LIN {X 0,Y 340.7,Z 163.546,A -85,B 0,C 180,E1 -14251.044,E2 -14251.044} C_VEL
LIN {X 0,Y 340.714,Z 163.527,A -85,B 0,C 180,E1 -14255.278,E2 -14255.278} C_VEL
LIN {X 0,Y 340.707,Z 163.544,A -85,B 0,C 180,E1 -14258.386,E2 -14258.386} C_VEL
LIN {X 0,Y 340.694,Z 163.543,A -85,B 0,C 180,E1 -14262.045,E2 -14262.045} C_VEL
LIN {X 0,Y 340.679,Z 163.532,A -85,B 0,C 180,E1 -14265.461,E2 -14265.461} C_VEL
LIN {X 0,Y 340.68,Z 163.504,A -85,B 0,C 180,E1 -14268.69,E2 -14268.69} C_VEL
LIN {X 0,Y 340.731,Z 163.543,A -85,B 0,C 180,E1 -14271.773,E2 -14271.773} C_VEL
LIN {X 0,Y 340.718,Z 163.515,A -85,B 0,C 180,E1 -14275.595,E2 -14275.595} C_VEL
LIN {X 0,Y 340.713,Z 163.54,A -85,B 0,C 180,E1 -14278.957,E2 -14278.957} C_VEL
LIN {X 0,Y 340.776,Z 163.536,A -85,B 0,C 180,E1 -14282.474,E2 -14282.474} C_VEL
LIN {X 0,Y 340.752,Z 163.541,A -85,B 0,C 180,E1 -14285.638,E2 -14285.638} C_VEL
LIN {X 0,Y 340.749,Z 163.652,A -85,B 0,C 180,E1 -14287.813,E2 -14287.813} C_VEL
LIN {X 0,Y 340.931,Z 164.489,A -85,B 0,C 180,E1 -14288.111,E2 -14288.111} C_VEL
LIN {X 0,Y 342.359,Z 167.226,A -85,B 0,C 180,E1 -14288.51,E2 -14288.51} C_VEL
LIN {X 0,Y 344.492,Z 169.253,A -85,B 0,C 180,E1 -14288.96,E2 -14288.96} C_VEL
LIN {X 0,Y 346.592,Z 172.469,A -85,B 0,C 180,E1 -14289.486,E2 -14289.486} C_VEL
LIN {X 0,Y 348.969,Z 174.84,A -85,B 0,C 180,E1 -14290.042,E2 -14290.042} C_VEL
LIN {X 0,Y 351.593,Z 178.193,A -85,B 0,C 180,E1 -14290.687,E2 -14290.687} C_VEL
LIN {X 0,Y 353.9,Z 180.47,A -85,B 0,C 180,E1 -14291.279,E2 -14291.279} C_VEL
LIN {X 0,Y 357.171,Z 184.318,A -85,B 0,C 180,E1 -14292.137,E2 -14292.137} C_VEL
LIN {X 0,Y 359.47,Z 186.421,A -85,B 0,C 180,E1 -14292.775,E2 -14292.775} C_VEL
LIN {X 0,Y 362.801,Z 190.102,A -85,B 0,C 180,E1 -14293.735,E2 -14293.735} C_VEL
LIN {X 0,Y 365.831,Z 192.588,A -85,B 0,C 180,E1 -14294.642,E2 -14294.642} C_VEL
LIN {X 0,Y 369.17,Z 196.334,A -85,B 0,C 180,E1 -14295.766,E2 -14295.766} C_VEL
LIN {X 0,Y 372.825,Z 199.259,A -85,B 0,C 180,E1 -14297.046,E2 -14297.046} C_VEL
LIN {X 0,Y 376.097,Z 202.708,A -85,B 0,C 180,E1 -14298.351,E2 -14298.351} C_VEL
LIN {X 0,Y 379.345,Z 205.079,A -85,B 0,C 180,E1 -14299.761,E2 -14299.761} C_VEL
LIN {X 0,Y 381.145,Z 206.14,A -85,B 0,C 180,E1 -14300.617,E2 -14300.617} C_VEL
LIN {X 0,Y 383.823,Z 209.323,A -85,B 0,C 180,E1 -14302.189,E2 -14302.189} C_VEL
LIN {X 0,Y 386.503,Z 211.375,A -85,B 0,C 180,E1 -14304.061,E2 -14304.061} C_VEL
LIN {X 0,Y 388.386,Z 212.415,A -85,B 0,C 180,E1 -14305.849,E2 -14305.849} C_VEL
LIN {X 0,Y 389.529,Z 212.797,A -85,B 0,C 180,E1 -14307.434,E2 -14307.434} C_VEL
LIN {X 0,Y 390.1,Z 213.221,A -85,B 0,C 180,E1 -14308.968,E2 -14308.968} C_VEL
LIN {X 0,Y 390.27,Z 213.15,A -85,B 0,C 180,E1 -14310,E2 -14310} C_VEL
LIN {X 0,Y 389.992,Z 213.112,A -85,B 0,C 180,E1 -14311.549,E2 -14311.549} C_VEL
LIN {X 0,Y 389.238,Z 212.653,A -85,B 0,C 180,E1 -14313.105,E2 -14313.105} C_VEL
LIN {X 0,Y 387.614,Z 212.058,A -85,B 0,C 180,E1 -14314.941,E2 -14314.941} C_VEL
LIN {X 0,Y 385.473,Z 210.702,A -85,B 0,C 180,E1 -14316.684,E2 -14316.684} C_VEL
LIN {X 0,Y 383.115,Z 208.634,A -85,B 0,C 180,E1 -14318.226,E2 -14318.226} C_VEL
LIN {X 0,Y 380.545,Z 205.669,A -85,B 0,C 180,E1 -14319.669,E2 -14319.669} C_VEL
LIN {X 0,Y 377.535,Z 203.906,A -85,B 0,C 180,E1 -14321.039,E2 -14321.039} C_VEL
LIN {X 0,Y 374.063,Z 200.682,A -85,B 0,C 180,E1 -14322.478,E2 -14322.478} C_VEL
LIN {X 0,Y 371.999,Z 198.446,A -85,B 0,C 180,E1 -14323.274,E2 -14323.274} C_VEL
LIN {X 0,Y 368.238,Z 195.449,A -85,B 0,C 180,E1 -14324.55,E2 -14324.55} C_VEL
LIN {X 0,Y 364.871,Z 191.735,A -85,B 0,C 180,E1 -14325.644,E2 -14325.644} C_VEL
LIN {X 0,Y 361.202,Z 188.491,A -85,B 0,C 180,E1 -14326.737,E2 -14326.737} C_VEL
LIN {X 0,Y 358.551,Z 185.445,A -85,B 0,C 180,E1 -14327.482,E2 -14327.482} C_VEL
LIN {X 0,Y 355.376,Z 182.455,A -85,B 0,C 180,E1 -14328.333,E2 -14328.333} C_VEL
LIN {X 0,Y 353.051,Z 179.523,A -85,B 0,C 180,E1 -14328.94,E2 -14328.94} C_VEL
LIN {X 0,Y 350.001,Z 176.372,A -85,B 0,C 180,E1 -14329.706,E2 -14329.706} C_VEL
LIN {X 0,Y 348.215,Z 173.968,A -85,B 0,C 180,E1 -14330.137,E2 -14330.137} C_VEL
LIN {X 0,Y 345.498,Z 171.058,A -85,B 0,C 180,E1 -14330.785,E2 -14330.785} C_VEL
LIN {X 0,Y 344.014,Z 168.683,A -85,B 0,C 180,E1 -14331.145,E2 -14331.145} C_VEL
LIN {X 0,Y 341.721,Z 166.358,A -85,B 0,C 180,E1 -14331.634,E2 -14331.634} C_VEL
LIN {X 0,Y 340.82,Z 164.079,A -85,B 0,C 180,E1 -14331.984,E2 -14331.984} C_VEL
LIN {X 0,Y 340.742,Z 163.555,A -85,B 0,C 180,E1 -14332.43,E2 -14332.43} C_VEL
LIN {X 0,Y 340.769,Z 163.54,A -85,B 0,C 180,E1 -14335.664,E2 -14335.664} C_VEL
LIN {X 0,Y 340.738,Z 163.528,A -85,B 0,C 180,E1 -14338.32,E2 -14338.32} C_VEL
LIN {X 0,Y 340.713,Z 163.54,A -85,B 0,C 180,E1 -14341.043,E2 -14341.043} C_VEL
LIN {X 0,Y 340.714,Z 163.517,A -85,B 0,C 180,E1 -14345.279,E2 -14345.279} C_VEL
LIN {X 0,Y 340.708,Z 163.547,A -85,B 0,C 180,E1 -14348.387,E2 -14348.387} C_VEL
LIN {X 0,Y 340.694,Z 163.499,A -85,B 0,C 180,E1 -14352.046,E2 -14352.046} C_VEL
LIN {X 0,Y 340.68,Z 163.546,A -85,B 0,C 180,E1 -14355.462,E2 -14355.462} C_VEL
LIN {X 0,Y 340.681,Z 163.536,A -85,B 0,C 180,E1 -14358.691,E2 -14358.691} C_VEL
LIN {X 0,Y 340.731,Z 163.541,A -85,B 0,C 180,E1 -14361.773,E2 -14361.773} C_VEL
LIN {X 0,Y 340.718,Z 163.522,A -85,B 0,C 180,E1 -14365.596,E2 -14365.596} C_VEL
LIN {X 0,Y 340.718,Z 163.542,A -85,B 0,C 180,E1 -14369.553,E2 -14369.553} C_VEL
LIN {X 0,Y 340.801,Z 163.511,A -85,B 0,C 180,E1 -14373.02,E2 -14373.02} C_VEL
LIN {X 0,Y 340.757,Z 163.528,A -85,B 0,C 180,E1 -14374.679,E2 -14374.679} C_VEL
LIN {X 0,Y 340.074,Z 163.621,A -85,B 0,C 180,E1 -14375.666,E2 -14375.666} C_VEL
LIN {X 0,Y 337.18,Z 163.982,A -85,B 0,C 180,E1 -14377.27,E2 -14377.27} C_VEL
LIN {X 0,Y 334.758,Z 164.276,A -85,B 0,C 180,E1 -14378.57,E2 -14378.57} C_VEL
LIN {X 0,Y 333.758,Z 164.391,A -85,B 0,C 180,E1 -14379.577,E2 -14379.577} C_VEL
LIN {X 0,Y 333.697,Z 164.392,A -85,B 0,C 180,E1 -14379.917,E2 -14379.917} C_VEL
LIN {X 0,Y 333.743,Z 164.401,A -85,B 0,C 180,E1 -14382.854,E2 -14382.854} C_VEL
LIN {X 0,Y 333.793,Z 164.402,A -85,B 0,C 180,E1 -14386.609,E2 -14386.609} C_VEL
LIN {X 0,Y 333.859,Z 164.366,A -85,B 0,C 180,E1 -14390.306,E2 -14390.306} C_VEL
LIN {X 0,Y 334.023,Z 164.369,A -85,B 0,C 180,E1 -14392.748,E2 -14392.748} C_VEL
LIN {X 0,Y 333.808,Z 164.403,A -85,B 0,C 180,E1 -14395.17,E2 -14395.17} C_VEL
LIN {X 0,Y 334.104,Z 164.352,A -85,B 0,C 180,E1 -14397.589,E2 -14397.589} C_VEL
LIN {X 0,Y 334.224,Z 164.319,A -85,B 0,C 180,E1 -14400.001,E2 -14400.001} C_VEL
LIN {X 0,Y 334.102,Z 164.359,A -85,B 0,C 180,E1 -14402.412,E2 -14402.412} C_VEL
LIN {X 0,Y 334.013,Z 164.374,A -85,B 0,C 180,E1 -14406.04,E2 -14406.04} C_VEL
LIN {X 0,Y 333.956,Z 164.361,A -85,B 0,C 180,E1 -14408.472,E2 -14408.472} C_VEL
LIN {X 0,Y 333.789,Z 164.397,A -85,B 0,C 180,E1 -14412.155,E2 -14412.155} C_VEL
LIN {X 0,Y 333.776,Z 164.399,A -85,B 0,C 180,E1 -14415.887,E2 -14415.887} C_VEL
LIN {X 0,Y 333.794,Z 164.375,A -85,B 0,C 180,E1 -14418.655,E2 -14418.655} C_VEL
LIN {X 0,Y 333.691,Z 164.414,A -85,B 0,C 180,E1 -14422.279,E2 -14422.279} C_VEL
LIN {X 0,Y 333.734,Z 164.392,A -85,B 0,C 180,E1 -14426.247,E2 -14426.247} C_VEL
LIN {X 0,Y 333.689,Z 164.41,A -85,B 0,C 180,E1 -14428.975,E2 -14428.975} C_VEL
LIN {X 0,Y 333.643,Z 164.416,A -85,B 0,C 180,E1 -14432.588,E2 -14432.588} C_VEL
LIN {X 0,Y 333.675,Z 164.415,A -85,B 0,C 180,E1 -14436.14,E2 -14436.14} C_VEL
LIN {X 0,Y 333.646,Z 164.414,A -85,B 0,C 180,E1 -14439.193,E2 -14439.193} C_VEL
LIN {X 0,Y 333.633,Z 164.429,A -85,B 0,C 180,E1 -14442.501,E2 -14442.501} C_VEL
LIN {X 0,Y 333.597,Z 164.429,A -85,B 0,C 180,E1 -14445.956,E2 -14445.956} C_VEL
LIN {X 0,Y 333.648,Z 164.399,A -85,B 0,C 180,E1 -14449.316,E2 -14449.316} C_VEL
LIN {X 0,Y 333.668,Z 164.417,A -85,B 0,C 180,E1 -14453.168,E2 -14453.168} C_VEL
LIN {X 0,Y 333.7,Z 164.494,A -85,B 0,C 180,E1 -14456.885,E2 -14456.885} C_VEL
LIN {X 0,Y 334.992,Z 170.834,A -85,B 0,C 180,E1 -14459.336,E2 -14459.336} C_VEL
LIN {X 0,Y 336.87,Z 180.369,A -85,B 0,C 180,E1 -14462.679,E2 -14462.679} C_VEL
LIN {X 0,Y 336.984,Z 184.304,A -85,B 0,C 180,E1 -14464.026,E2 -14464.026} C_VEL
LIN {X 0,Y 336.226,Z 190.3,A -85,B 0,C 180,E1 -14465.935,E2 -14465.935} C_VEL
LIN {X 0,Y 338.132,Z 199.11,A -85,B 0,C 180,E1 -14466.325,E2 -14466.325} C_VEL
LIN {X 0,Y 343.281,Z 226.363,A -85,B 0,C 180,E1 -14467.304,E2 -14467.304} C_VEL
LIN {X 0,Y 343.746,Z 230.733,A -85,B 0,C 180,E1 -14467.433,E2 -14467.433} C_VEL
LIN {X 0,Y 342.36,Z 296.356,A -85,B 0,C 180,E1 -14468.828,E2 -14468.828} C_VEL
LIN {X 0,Y 341.833,Z 306.667,A -85,B 0,C 180,E1 -14469.189,E2 -14469.189} C_VEL
LIN {X 0,Y 341.14,Z 316.179,A -85,B 0,C 180,E1 -14469.657,E2 -14469.657} C_VEL
LIN {X 0,Y 340.356,Z 325.253,A -85,B 0,C 180,E1 -14470.237,E2 -14470.237} C_VEL
LIN {X 0,Y 339.426,Z 334.384,A -85,B 0,C 180,E1 -14470.967,E2 -14470.967} C_VEL
LIN {X 0,Y 338.346,Z 343.378,A -85,B 0,C 180,E1 -14471.846,E2 -14471.846} C_VEL
LIN {X 0,Y 337.268,Z 352.105,A -85,B 0,C 180,E1 -14472.882,E2 -14472.882} C_VEL
LIN {X 0,Y 336.235,Z 360.291,A -85,B 0,C 180,E1 -14474.05,E2 -14474.05} C_VEL
LIN {X 0,Y 335.224,Z 368.347,A -85,B 0,C 180,E1 -14475.429,E2 -14475.429} C_VEL
LIN {X 0,Y 334.464,Z 374.299,A -85,B 0,C 180,E1 -14476.636,E2 -14476.636} C_VEL
LIN {X 0,Y 333.583,Z 380.614,A -85,B 0,C 180,E1 -14478.146,E2 -14478.146} C_VEL
LIN {X 0,Y 332.98,Z 385.877,A -85,B 0,C 180,E1 -14479.665,E2 -14479.665} C_VEL
LIN {X 0,Y 332.46,Z 391.008,A -85,B 0,C 180,E1 -14481.49,E2 -14481.49} C_VEL
LIN {X 0,Y 332.124,Z 394.996,A -85,B 0,C 180,E1 -14483.317,E2 -14483.317} C_VEL
LIN {X 0,Y 331.973,Z 397.946,A -85,B 0,C 180,E1 -14485.142,E2 -14485.142} C_VEL
LIN {X 0,Y 331.916,Z 400.393,A -85,B 0,C 180,E1 -14487.573,E2 -14487.573} C_VEL
LIN {X 0,Y 331.913,Z 400.982,A -85,B 0,C 180,E1 -14488.787,E2 -14488.787} C_VEL
LIN {X 0,Y 331.913,Z 400.982,A -85,B 0,C 180,E1 -14491.213,E2 -14491.213} C_VEL
LIN {X 0,Y 331.916,Z 400.393,A -85,B 0,C 180,E1 -14492.427,E2 -14492.427} C_VEL
LIN {X 0,Y 331.971,Z 397.946,A -85,B 0,C 180,E1 -14494.858,E2 -14494.858} C_VEL
LIN {X 0,Y 332.105,Z 394.996,A -85,B 0,C 180,E1 -14496.684,E2 -14496.684} C_VEL
LIN {X 0,Y 332.46,Z 391.008,A -85,B 0,C 180,E1 -14498.51,E2 -14498.51} C_VEL
LIN {X 0,Y 332.98,Z 385.877,A -85,B 0,C 180,E1 -14500.335,E2 -14500.335} C_VEL
LIN {X 0,Y 333.582,Z 380.614,A -85,B 0,C 180,E1 -14501.854,E2 -14501.854} C_VEL
LIN {X 0,Y 334.472,Z 374.299,A -85,B 0,C 180,E1 -14503.364,E2 -14503.364} C_VEL
LIN {X 0,Y 335.216,Z 368.347,A -85,B 0,C 180,E1 -14504.571,E2 -14504.571} C_VEL
LIN {X 0,Y 336.147,Z 361.42,A -85,B 0,C 180,E1 -14505.771,E2 -14505.771} C_VEL
LIN {X 0,Y 337.152,Z 353.24,A -85,B 0,C 180,E1 -14506.967,E2 -14506.967} C_VEL
LIN {X 0,Y 338.201,Z 344.73,A -85,B 0,C 180,E1 -14508.005,E2 -14508.005} C_VEL
LIN {X 0,Y 339.229,Z 336.016,A -85,B 0,C 180,E1 -14508.887,E2 -14508.887} C_VEL
LIN {X 0,Y 340.282,Z 326.26,A -85,B 0,C 180,E1 -14509.688,E2 -14509.688} C_VEL
LIN {X 0,Y 341.126,Z 316.179,A -85,B 0,C 180,E1 -14510.344,E2 -14510.344} C_VEL
LIN {X 0,Y 341.811,Z 306.666,A -85,B 0,C 180,E1 -14510.813,E2 -14510.813} C_VEL
LIN {X 0,Y 342.383,Z 296.357,A -85,B 0,C 180,E1 -14511.17,E2 -14511.17} C_VEL
LIN {X 0,Y 343.642,Z 228.699,A -85,B 0,C 180,E1 -14512.619,E2 -14512.619} C_VEL
LIN {X 0,Y 338.791,Z 202.108,A -85,B 0,C 180,E1 -14513.558,E2 -14513.558} C_VEL
LIN {X 0,Y 336.246,Z 190.61,A -85,B 0,C 180,E1 -14514.031,E2 -14514.031} C_VEL
LIN {X 0,Y 336.329,Z 189.001,A -85,B 0,C 180,E1 -14514.407,E2 -14514.407} C_VEL
LIN {X 0,Y 337.122,Z 183.29,A -85,B 0,C 180,E1 -14516.307,E2 -14516.307} C_VEL
LIN {X 0,Y 336.53,Z 178.586,A -85,B 0,C 180,E1 -14517.959,E2 -14517.959} C_VEL
LIN {X 0,Y 334.839,Z 169.883,A -85,B 0,C 180,E1 -14521.091,E2 -14521.091} C_VEL
LIN {X 0,Y 333.674,Z 164.43,A -85,B 0,C 180,E1 -14523.204,E2 -14523.204} C_VEL
LIN {X 0,Y 333.668,Z 164.417,A -85,B 0,C 180,E1 -14526.832,E2 -14526.832} C_VEL
LIN {X 0,Y 333.647,Z 164.399,A -85,B 0,C 180,E1 -14530.767,E2 -14530.767} C_VEL
LIN {X 0,Y 333.593,Z 164.428,A -85,B 0,C 180,E1 -14534.25,E2 -14534.25} C_VEL
LIN {X 0,Y 333.642,Z 164.428,A -85,B 0,C 180,E1 -14537.618,E2 -14537.618} C_VEL
LIN {X 0,Y 333.652,Z 164.416,A -85,B 0,C 180,E1 -14541.201,E2 -14541.201} C_VEL
LIN {X 0,Y 333.675,Z 164.415,A -85,B 0,C 180,E1 -14543.86,E2 -14543.86} C_VEL
LIN {X 0,Y 333.643,Z 164.416,A -85,B 0,C 180,E1 -14547.412,E2 -14547.412} C_VEL
LIN {X 0,Y 333.689,Z 164.41,A -85,B 0,C 180,E1 -14551.025,E2 -14551.025} C_VEL
LIN {X 0,Y 333.734,Z 164.392,A -85,B 0,C 180,E1 -14553.753,E2 -14553.753} C_VEL
LIN {X 0,Y 333.718,Z 164.411,A -85,B 0,C 180,E1 -14557.913,E2 -14557.913} C_VEL
LIN {X 0,Y 333.792,Z 164.376,A -85,B 0,C 180,E1 -14561.589,E2 -14561.589} C_VEL
LIN {X 0,Y 333.807,Z 164.401,A -85,B 0,C 180,E1 -14565.576,E2 -14565.576} C_VEL
LIN {X 0,Y 333.831,Z 164.375,A -85,B 0,C 180,E1 -14569.077,E2 -14569.077} C_VEL
LIN {X 0,Y 334.005,Z 164.366,A -85,B 0,C 180,E1 -14572.746,E2 -14572.746} C_VEL
LIN {X 0,Y 333.807,Z 164.403,A -85,B 0,C 180,E1 -14575.168,E2 -14575.168} C_VEL
LIN {X 0,Y 334.102,Z 164.359,A -85,B 0,C 180,E1 -14577.588,E2 -14577.588} C_VEL
LIN {X 0,Y 334.224,Z 164.319,A -85,B 0,C 180,E1 -14579.999,E2 -14579.999} C_VEL
LIN {X 0,Y 334.104,Z 164.352,A -85,B 0,C 180,E1 -14582.411,E2 -14582.411} C_VEL
LIN {X 0,Y 334.023,Z 164.369,A -85,B 0,C 180,E1 -14587.252,E2 -14587.252} C_VEL
LIN {X 0,Y 333.83,Z 164.376,A -85,B 0,C 180,E1 -14590.921,E2 -14590.921} C_VEL
LIN {X 0,Y 333.805,Z 164.404,A -85,B 0,C 180,E1 -14594.634,E2 -14594.634} C_VEL
LIN {X 0,Y 333.792,Z 164.376,A -85,B 0,C 180,E1 -14598.654,E2 -14598.654} C_VEL
LIN {X 0,Y 333.688,Z 164.419,A -85,B 0,C 180,E1 -14602.278,E2 -14602.278} C_VEL
LIN {X 0,Y 333.732,Z 164.395,A -85,B 0,C 180,E1 -14606.246,E2 -14606.246} C_VEL
LIN {X 0,Y 333.707,Z 164.406,A -85,B 0,C 180,E1 -14608.972,E2 -14608.972} C_VEL
LIN {X 0,Y 333.639,Z 164.421,A -85,B 0,C 180,E1 -14612.587,E2 -14612.587} C_VEL
LIN {X 0,Y 333.673,Z 164.417,A -85,B 0,C 180,E1 -14616.138,E2 -14616.138} C_VEL
LIN {X 0,Y 333.642,Z 164.419,A -85,B 0,C 180,E1 -14619.192,E2 -14619.192} C_VEL
LIN {X 0,Y 333.629,Z 164.424,A -85,B 0,C 180,E1 -14622.5,E2 -14622.5} C_VEL
LIN {X 0,Y 333.617,Z 164.404,A -85,B 0,C 180,E1 -14625.959,E2 -14625.959} C_VEL
LIN {X 0,Y 333.642,Z 164.388,A -85,B 0,C 180,E1 -14629.315,E2 -14629.315} C_VEL
LIN {X 0,Y 333.662,Z 164.416,A -85,B 0,C 180,E1 -14633.167,E2 -14633.167} C_VEL
LIN {X 0,Y 333.638,Z 164.409,A -85,B 0,C 180,E1 -14636.792,E2 -14636.792} C_VEL
LIN {X 0,Y 333.7,Z 164.403,A -85,B 0,C 180,E1 -14639.71,E2 -14639.71} C_VEL
LIN {X 0,Y 333.74,Z 164.411,A -85,B 0,C 180,E1 -14642.401,E2 -14642.401} C_VEL
LIN {X 0,Y 333.723,Z 164.417,A -85,B 0,C 180,E1 -14645.091,E2 -14645.091} C_VEL
LIN {X 0,Y 333.714,Z 164.564,A -85,B 0,C 180,E1 -14646.635,E2 -14646.635} C_VEL
LIN {X 0,Y 333.902,Z 165.477,A -85,B 0,C 180,E1 -14646.906,E2 -14646.906} C_VEL
LIN {X 0,Y 335.44,Z 168.254,A -85,B 0,C 180,E1 -14647.293,E2 -14647.293} C_VEL
LIN {X 0,Y 337.24,Z 170.143,A -85,B 0,C 180,E1 -14647.649,E2 -14647.649} C_VEL
LIN {X 0,Y 339.606,Z 173.544,A -85,B 0,C 180,E1 -14648.193,E2 -14648.193} C_VEL
LIN {X 0,Y 341.244,Z 175.293,A -85,B 0,C 180,E1 -14648.55,E2 -14648.55} C_VEL
LIN {X 0,Y 344.183,Z 179.022,A -85,B 0,C 180,E1 -14649.205,E2 -14649.205} C_VEL
LIN {X 0,Y 346.131,Z 181.092,A -85,B 0,C 180,E1 -14649.669,E2 -14649.669} C_VEL
LIN {X 0,Y 349.588,Z 185.013,A -85,B 0,C 180,E1 -14650.485,E2 -14650.485} C_VEL
LIN {X 0,Y 351.431,Z 186.973,A -85,B 0,C 180,E1 -14650.949,E2 -14650.949} C_VEL
LIN {X 0,Y 355.263,Z 191.068,A -85,B 0,C 180,E1 -14651.929,E2 -14651.929} C_VEL
LIN {X 0,Y 357.233,Z 192.994,A -85,B 0,C 180,E1 -14652.464,E2 -14652.464} C_VEL
LIN {X 0,Y 361.224,Z 197.042,A -85,B 0,C 180,E1 -14653.582,E2 -14653.582} C_VEL
LIN {X 0,Y 363.73,Z 199.166,A -85,B 0,C 180,E1 -14654.333,E2 -14654.333} C_VEL
LIN {X 0,Y 367.349,Z 202.937,A -85,B 0,C 180,E1 -14655.493,E2 -14655.493} C_VEL
LIN {X 0,Y 371.23,Z 206.057,A -85,B 0,C 180,E1 -14656.813,E2 -14656.813} C_VEL
LIN {X 0,Y 374.708,Z 209.566,A -85,B 0,C 180,E1 -14658.165,E2 -14658.165} C_VEL
LIN {X 0,Y 378.246,Z 212.061,A -85,B 0,C 180,E1 -14659.673,E2 -14659.673} C_VEL
LIN {X 0,Y 379.883,Z 213.156,A -85,B 0,C 180,E1 -14660.464,E2 -14660.464} C_VEL
LIN {X 0,Y 382.521,Z 216.119,A -85,B 0,C 180,E1 -14661.961,E2 -14661.961} C_VEL
LIN {X 0,Y 384.968,Z 218.058,A -85,B 0,C 180,E1 -14663.58,E2 -14663.58} C_VEL
LIN {X 0,Y 387.279,Z 219.357,A -85,B 0,C 180,E1 -14665.577,E2 -14665.577} C_VEL
LIN {X 0,Y 388.665,Z 219.823,A -85,B 0,C 180,E1 -14667.428,E2 -14667.428} C_VEL
LIN {X 0,Y 389.239,Z 220.26,A -85,B 0,C 180,E1 -14668.965,E2 -14668.965} C_VEL
LIN {X 0,Y 389.407,Z 220.18,A -85,B 0,C 180,E1 -14670,E2 -14670} C_VEL
LIN {X 0,Y 389.126,Z 220.135,A -85,B 0,C 180,E1 -14671.552,E2 -14671.552} C_VEL
LIN {X 0,Y 388.361,Z 219.7,A -85,B 0,C 180,E1 -14673.112,E2 -14673.112} C_VEL
LIN {X 0,Y 386.736,Z 219.095,A -85,B 0,C 180,E1 -14674.943,E2 -14674.943} C_VEL
LIN {X 0,Y 384.56,Z 217.784,A -85,B 0,C 180,E1 -14676.7,E2 -14676.7} C_VEL
LIN {X 0,Y 382.058,Z 215.691,A -85,B 0,C 180,E1 -14678.309,E2 -14678.309} C_VEL
LIN {X 0,Y 379.214,Z 212.563,A -85,B 0,C 180,E1 -14679.864,E2 -14679.864} C_VEL
LIN {X 0,Y 375.944,Z 210.617,A -85,B 0,C 180,E1 -14681.308,E2 -14681.308} C_VEL
LIN {X 0,Y 372.666,Z 207.666,A -85,B 0,C 180,E1 -14682.629,E2 -14682.629} C_VEL
LIN {X 0,Y 370.003,Z 204.947,A -85,B 0,C 180,E1 -14683.635,E2 -14683.635} C_VEL
LIN {X 0,Y 365.741,Z 201.421,A -85,B 0,C 180,E1 -14685.038,E2 -14685.038} C_VEL
LIN {X 0,Y 362.655,Z 198.154,A -85,B 0,C 180,E1 -14685.995,E2 -14685.995} C_VEL
LIN {X 0,Y 358.732,Z 194.722,A -85,B 0,C 180,E1 -14687.109,E2 -14687.109} C_VEL
LIN {X 0,Y 355.812,Z 191.514,A -85,B 0,C 180,E1 -14687.928,E2 -14687.928} C_VEL
LIN {X 0,Y 352.19,Z 187.976,A -85,B 0,C 180,E1 -14688.848,E2 -14688.848} C_VEL
LIN {X 0,Y 350.013,Z 185.387,A -85,B 0,C 180,E1 -14689.415,E2 -14689.415} C_VEL
LIN {X 0,Y 346.374,Z 181.474,A -85,B 0,C 180,E1 -14690.27,E2 -14690.27} C_VEL
LIN {X 0,Y 344.964,Z 179.746,A -85,B 0,C 180,E1 -14690.614,E2 -14690.614} C_VEL
LIN {X 0,Y 341.952,Z 176.423,A -85,B 0,C 180,E1 -14691.286,E2 -14691.286} C_VEL
LIN {X 0,Y 340.286,Z 174.152,A -85,B 0,C 180,E1 -14691.662,E2 -14691.662} C_VEL
LIN {X 0,Y 337.9,Z 171.309,A -85,B 0,C 180,E1 -14692.197,E2 -14692.197} C_VEL
LIN {X 0,Y 336.543,Z 169.281,A -85,B 0,C 180,E1 -14692.493,E2 -14692.493} C_VEL
LIN {X 0,Y 334.617,Z 167.13,A -85,B 0,C 180,E1 -14692.878,E2 -14692.878} C_VEL
LIN {X 0,Y 333.802,Z 165.071,A -85,B 0,C 180,E1 -14693.171,E2 -14693.171} C_VEL
LIN {X 0,Y 333.68,Z 164.493,A -85,B 0,C 180,E1 -14693.425,E2 -14693.425} C_VEL
LIN {X 0,Y 333.732,Z 164.416,A -85,B 0,C 180,E1 -14696.246,E2 -14696.246} C_VEL
LIN {X 0,Y 333.708,Z 164.397,A -85,B 0,C 180,E1 -14698.972,E2 -14698.972} C_VEL
LIN {X 0,Y 333.648,Z 164.418,A -85,B 0,C 180,E1 -14702.589,E2 -14702.589} C_VEL
LIN {X 0,Y 333.673,Z 164.405,A -85,B 0,C 180,E1 -14706.139,E2 -14706.139} C_VEL
LIN {X 0,Y 333.643,Z 164.418,A -85,B 0,C 180,E1 -14709.192,E2 -14709.192} C_VEL
LIN {X 0,Y 333.628,Z 164.379,A -85,B 0,C 180,E1 -14712.5,E2 -14712.5} C_VEL
LIN {X 0,Y 333.617,Z 164.426,A -85,B 0,C 180,E1 -14715.959,E2 -14715.959} C_VEL
LIN {X 0,Y 333.642,Z 164.41,A -85,B 0,C 180,E1 -14719.316,E2 -14719.316} C_VEL
LIN {X 0,Y 333.662,Z 164.42,A -85,B 0,C 180,E1 -14723.168,E2 -14723.168} C_VEL
LIN {X 0,Y 333.669,Z 164.4,A -85,B 0,C 180,E1 -14725.342,E2 -14725.342} C_VEL
LIN {X 0,Y 333.698,Z 164.417,A -85,B 0,C 180,E1 -14729.711,E2 -14729.711} C_VEL
LIN {X 0,Y 333.74,Z 164.39,A -85,B 0,C 180,E1 -14732.402,E2 -14732.402} C_VEL
LIN {X 0,Y 333.723,Z 164.411,A -85,B 0,C 180,E1 -14735.091,E2 -14735.091} C_VEL
LIN {X 0,Y 333.676,Z 164.409,A -85,B 0,C 180,E1 -14739.02,E2 -14739.02} C_VEL
LIN {X 0,Y 333.697,Z 164.392,A -85,B 0,C 180,E1 -14739.917,E2 -14739.917} C_VEL
LIN {X 0,Y 333.086,Z 164.465,A -85,B 0,C 180,E1 -14740.925,E2 -14740.925} C_VEL
LIN {X 0,Y 330.263,Z 164.828,A -85,B 0,C 180,E1 -14742.564,E2 -14742.564} C_VEL
LIN {X 0,Y 327.849,Z 165.141,A -85,B 0,C 180,E1 -14743.892,E2 -14743.892} C_VEL
LIN {X 0,Y 326.827,Z 165.273,A -85,B 0,C 180,E1 -14744.92,E2 -14744.92} C_VEL
LIN {X 0,Y 326.754,Z 165.282,A -85,B 0,C 180,E1 -14745.268,E2 -14745.268} C_VEL
LIN {X 0,Y 326.766,Z 165.259,A -85,B 0,C 180,E1 -14748.84,E2 -14748.84} C_VEL
LIN {X 0,Y 326.974,Z 165.247,A -85,B 0,C 180,E1 -14752.591,E2 -14752.591} C_VEL
LIN {X 0,Y 326.775,Z 165.279,A -85,B 0,C 180,E1 -14755.066,E2 -14755.066} C_VEL
LIN {X 0,Y 327.045,Z 165.231,A -85,B 0,C 180,E1 -14757.537,E2 -14757.537} C_VEL
LIN {X 0,Y 327.175,Z 165.196,A -85,B 0,C 180,E1 -14760.001,E2 -14760.001} C_VEL
LIN {X 0,Y 327.043,Z 165.238,A -85,B 0,C 180,E1 -14762.464,E2 -14762.464} C_VEL
LIN {X 0,Y 326.988,Z 165.248,A -85,B 0,C 180,E1 -14766.17,E2 -14766.17} C_VEL
LIN {X 0,Y 326.803,Z 165.243,A -85,B 0,C 180,E1 -14769.907,E2 -14769.907} C_VEL
LIN {X 0,Y 326.757,Z 165.28,A -85,B 0,C 180,E1 -14773.686,E2 -14773.686} C_VEL
LIN {X 0,Y 326.697,Z 165.264,A -85,B 0,C 180,E1 -14777.529,E2 -14777.529} C_VEL
LIN {X 0,Y 326.661,Z 165.275,A -85,B 0,C 180,E1 -14780.136,E2 -14780.136} C_VEL
LIN {X 0,Y 326.651,Z 165.291,A -85,B 0,C 180,E1 -14784.13,E2 -14784.13} C_VEL
LIN {X 0,Y 326.682,Z 165.267,A -85,B 0,C 180,E1 -14786.859,E2 -14786.859} C_VEL
LIN {X 0,Y 326.633,Z 165.299,A -85,B 0,C 180,E1 -14790.61,E2 -14790.61} C_VEL
LIN {X 0,Y 326.606,Z 165.281,A -85,B 0,C 180,E1 -14794.02,E2 -14794.02} C_VEL
LIN {X 0,Y 326.627,Z 165.299,A -85,B 0,C 180,E1 -14797.239,E2 -14797.239} C_VEL
LIN {X 0,Y 326.578,Z 165.298,A -85,B 0,C 180,E1 -14801.132,E2 -14801.132} C_VEL
LIN {X 0,Y 326.527,Z 165.303,A -85,B 0,C 180,E1 -14804.743,E2 -14804.743} C_VEL
LIN {X 0,Y 326.577,Z 165.292,A -85,B 0,C 180,E1 -14808.155,E2 -14808.155} C_VEL
LIN {X 0,Y 326.626,Z 165.289,A -85,B 0,C 180,E1 -14811.392,E2 -14811.392} C_VEL
LIN {X 0,Y 326.621,Z 165.284,A -85,B 0,C 180,E1 -14814.852,E2 -14814.852} C_VEL
LIN {X 0,Y 326.636,Z 165.412,A -85,B 0,C 180,E1 -14816.489,E2 -14816.489} C_VEL
LIN {X 0,Y 327.993,Z 171.946,A -85,B 0,C 180,E1 -14819.053,E2 -14819.053} C_VEL
LIN {X 0,Y 329.629,Z 180.163,A -85,B 0,C 180,E1 -14822.027,E2 -14822.027} C_VEL
LIN {X 0,Y 330.134,Z 184.112,A -85,B 0,C 180,E1 -14823.445,E2 -14823.445} C_VEL
LIN {X 0,Y 329.408,Z 189.966,A -85,B 0,C 180,E1 -14825.381,E2 -14825.381} C_VEL
LIN {X 0,Y 330.263,Z 194.285,A -85,B 0,C 180,E1 -14825.618,E2 -14825.618} C_VEL
LIN {X 0,Y 335.005,Z 217.321,A -85,B 0,C 180,E1 -14826.51,E2 -14826.51} C_VEL
LIN {X 0,Y 337.162,Z 230.559,A -85,B 0,C 180,E1 -14826.968,E2 -14826.968} C_VEL
LIN {X 0,Y 335.756,Z 296.164,A -85,B 0,C 180,E1 -14828.391,E2 -14828.391} C_VEL
LIN {X 0,Y 335.222,Z 306.475,A -85,B 0,C 180,E1 -14828.758,E2 -14828.758} C_VEL
LIN {X 0,Y 334.508,Z 315.988,A -85,B 0,C 180,E1 -14829.235,E2 -14829.235} C_VEL
LIN {X 0,Y 333.688,Z 325.061,A -85,B 0,C 180,E1 -14829.826,E2 -14829.826} C_VEL
LIN {X 0,Y 332.71,Z 334.193,A -85,B 0,C 180,E1 -14830.568,E2 -14830.568} C_VEL
LIN {X 0,Y 331.604,Z 343.186,A -85,B 0,C 180,E1 -14831.464,E2 -14831.464} C_VEL
LIN {X 0,Y 330.471,Z 351.913,A -85,B 0,C 180,E1 -14832.519,E2 -14832.519} C_VEL
LIN {X 0,Y 329.473,Z 359.673,A -85,B 0,C 180,E1 -14833.643,E2 -14833.643} C_VEL
LIN {X 0,Y 328.548,Z 366.662,A -85,B 0,C 180,E1 -14834.835,E2 -14834.835} C_VEL
LIN {X 0,Y 327.76,Z 372.731,A -85,B 0,C 180,E1 -14836.041,E2 -14836.041} C_VEL
LIN {X 0,Y 326.771,Z 379.266,A -85,B 0,C 180,E1 -14837.58,E2 -14837.58} C_VEL
LIN {X 0,Y 326.2,Z 383.768,A -85,B 0,C 180,E1 -14838.819,E2 -14838.819} C_VEL
LIN {X 0,Y 325.572,Z 389.261,A -85,B 0,C 180,E1 -14840.683,E2 -14840.683} C_VEL
LIN {X 0,Y 325.153,Z 393.587,A -85,B 0,C 180,E1 -14842.549,E2 -14842.549} C_VEL
LIN {X 0,Y 324.925,Z 396.619,A -85,B 0,C 180,E1 -14844.251,E2 -14844.251} C_VEL
LIN {X 0,Y 324.876,Z 399.144,A -85,B 0,C 180,E1 -14846.279,E2 -14846.279} C_VEL
LIN {X 0,Y 324.835,Z 400.202,A -85,B 0,C 180,E1 -14847.52,E2 -14847.52} C_VEL
LIN {X 0,Y 324.822,Z 400.791,A -85,B 0,C 180,E1 -14848.76,E2 -14848.76} C_VEL
LIN {X 0,Y 324.822,Z 400.791,A -85,B 0,C 180,E1 -14851.24,E2 -14851.24} C_VEL
LIN {X 0,Y 324.835,Z 400.202,A -85,B 0,C 180,E1 -14852.48,E2 -14852.48} C_VEL
LIN {X 0,Y 324.881,Z 397.754,A -85,B 0,C 180,E1 -14854.964,E2 -14854.964} C_VEL
LIN {X 0,Y 325.047,Z 394.804,A -85,B 0,C 180,E1 -14856.83,E2 -14856.83} C_VEL
LIN {X 0,Y 325.4,Z 390.815,A -85,B 0,C 180,E1 -14858.696,E2 -14858.696} C_VEL
LIN {X 0,Y 325.959,Z 385.684,A -85,B 0,C 180,E1 -14860.56,E2 -14860.56} C_VEL
LIN {X 0,Y 326.617,Z 380.422,A -85,B 0,C 180,E1 -14862.11,E2 -14862.11} C_VEL
LIN {X 0,Y 327.554,Z 374.107,A -85,B 0,C 180,E1 -14863.651,E2 -14863.651} C_VEL
LIN {X 0,Y 328.32,Z 368.154,A -85,B 0,C 180,E1 -14864.884,E2 -14864.884} C_VEL
LIN {X 0,Y 329.28,Z 361.228,A -85,B 0,C 180,E1 -14866.109,E2 -14866.109} C_VEL
LIN {X 0,Y 330.325,Z 353.047,A -85,B 0,C 180,E1 -14867.329,E2 -14867.329} C_VEL
LIN {X 0,Y 331.458,Z 344.538,A -85,B 0,C 180,E1 -14868.385,E2 -14868.385} C_VEL
LIN {X 0,Y 332.516,Z 335.824,A -85,B 0,C 180,E1 -14869.284,E2 -14869.284} C_VEL
LIN {X 0,Y 333.603,Z 326.068,A -85,B 0,C 180,E1 -14870.099,E2 -14870.099} C_VEL
LIN {X 0,Y 334.473,Z 315.987,A -85,B 0,C 180,E1 -14870.767,E2 -14870.767} C_VEL
LIN {X 0,Y 335.198,Z 306.475,A -85,B 0,C 180,E1 -14871.243,E2 -14871.243} C_VEL
LIN {X 0,Y 335.778,Z 296.165,A -85,B 0,C 180,E1 -14871.607,E2 -14871.607} C_VEL
LIN {X 0,Y 337.131,Z 230.29,A -85,B 0,C 180,E1 -14873.041,E2 -14873.041} C_VEL
LIN {X 0,Y 333.079,Z 207.235,A -85,B 0,C 180,E1 -14873.865,E2 -14873.865} C_VEL
LIN {X 0,Y 329.433,Z 190.195,A -85,B 0,C 180,E1 -14874.582,E2 -14874.582} C_VEL
LIN {X 0,Y 329.641,Z 187.957,A -85,B 0,C 180,E1 -14875.239,E2 -14875.239} C_VEL
LIN {X 0,Y 330.155,Z 183.942,A -85,B 0,C 180,E1 -14876.612,E2 -14876.612} C_VEL
LIN {X 0,Y 328.872,Z 176.177,A -85,B 0,C 180,E1 -14879.44,E2 -14879.44} C_VEL
LIN {X 0,Y 326.906,Z 166.644,A -85,B 0,C 180,E1 -14883.023,E2 -14883.023} C_VEL
LIN {X 0,Y 326.626,Z 165.314,A -85,B 0,C 180,E1 -14883.584,E2 -14883.584} C_VEL
LIN {X 0,Y 326.631,Z 165.298,A -85,B 0,C 180,E1 -14887.238,E2 -14887.238} C_VEL
LIN {X 0,Y 326.578,Z 165.282,A -85,B 0,C 180,E1 -14891.13,E2 -14891.13} C_VEL
LIN {X 0,Y 326.527,Z 165.306,A -85,B 0,C 180,E1 -14894.742,E2 -14894.742} C_VEL
LIN {X 0,Y 326.576,Z 165.304,A -85,B 0,C 180,E1 -14898.153,E2 -14898.153} C_VEL
LIN {X 0,Y 326.623,Z 165.294,A -85,B 0,C 180,E1 -14901.391,E2 -14901.391} C_VEL
LIN {X 0,Y 326.619,Z 165.286,A -85,B 0,C 180,E1 -14904.851,E2 -14904.851} C_VEL
LIN {X 0,Y 326.607,Z 165.292,A -85,B 0,C 180,E1 -14907.455,E2 -14907.455} C_VEL
LIN {X 0,Y 326.647,Z 165.294,A -85,B 0,C 180,E1 -14910.339,E2 -14910.339} C_VEL
LIN {X 0,Y 326.689,Z 165.275,A -85,B 0,C 180,E1 -14914.515,E2 -14914.515} C_VEL
LIN {X 0,Y 326.644,Z 165.29,A -85,B 0,C 180,E1 -14918.544,E2 -14918.544} C_VEL
LIN {X 0,Y 326.743,Z 165.252,A -85,B 0,C 180,E1 -14921.177,E2 -14921.177} C_VEL
LIN {X 0,Y 326.761,Z 165.279,A -85,B 0,C 180,E1 -14925.432,E2 -14925.432} C_VEL
LIN {X 0,Y 326.767,Z 165.257,A -85,B 0,C 180,E1 -14928.838,E2 -14928.838} C_VEL
LIN {X 0,Y 326.957,Z 165.242,A -85,B 0,C 180,E1 -14932.589,E2 -14932.589} C_VEL
LIN {X 0,Y 326.774,Z 165.28,A -85,B 0,C 180,E1 -14935.064,E2 -14935.064} C_VEL
LIN {X 0,Y 327.043,Z 165.238,A -85,B 0,C 180,E1 -14937.536,E2 -14937.536} C_VEL
LIN {X 0,Y 327.175,Z 165.196,A -85,B 0,C 180,E1 -14939.999,E2 -14939.999} C_VEL
LIN {X 0,Y 327.045,Z 165.231,A -85,B 0,C 180,E1 -14942.463,E2 -14942.463} C_VEL
LIN {X 0,Y 326.968,Z 165.249,A -85,B 0,C 180,E1 -14946.644,E2 -14946.644} C_VEL
LIN {X 0,Y 326.81,Z 165.243,A -85,B 0,C 180,E1 -14949.906,E2 -14949.906} C_VEL
LIN {X 0,Y 326.755,Z 165.28,A -85,B 0,C 180,E1 -14953.685,E2 -14953.685} C_VEL
LIN {X 0,Y 326.695,Z 165.271,A -85,B 0,C 180,E1 -14957.527,E2 -14957.527} C_VEL
LIN {X 0,Y 326.658,Z 165.27,A -85,B 0,C 180,E1 -14960.134,E2 -14960.134} C_VEL
LIN {X 0,Y 326.648,Z 165.294,A -85,B 0,C 180,E1 -14964.128,E2 -14964.128} C_VEL
LIN {X 0,Y 326.681,Z 165.269,A -85,B 0,C 180,E1 -14966.857,E2 -14966.857} C_VEL
LIN {X 0,Y 326.635,Z 165.297,A -85,B 0,C 180,E1 -14970.611,E2 -14970.611} C_VEL
LIN {X 0,Y 326.602,Z 165.281,A -85,B 0,C 180,E1 -14974.019,E2 -14974.019} C_VEL
LIN {X 0,Y 326.625,Z 165.3,A -85,B 0,C 180,E1 -14977.239,E2 -14977.239} C_VEL
LIN {X 0,Y 326.573,Z 165.291,A -85,B 0,C 180,E1 -14981.131,E2 -14981.131} C_VEL
LIN {X 0,Y 326.552,Z 165.301,A -85,B 0,C 180,E1 -14984.748,E2 -14984.748} C_VEL
LIN {X 0,Y 326.571,Z 165.256,A -85,B 0,C 180,E1 -14988.154,E2 -14988.154} C_VEL
LIN {X 0,Y 326.62,Z 165.3,A -85,B 0,C 180,E1 -14991.391,E2 -14991.391} C_VEL
LIN {X 0,Y 326.615,Z 165.271,A -85,B 0,C 180,E1 -14994.851,E2 -14994.851} C_VEL
LIN {X 0,Y 326.612,Z 165.295,A -85,B 0,C 180,E1 -14997.456,E2 -14997.456} C_VEL
LIN {X 0,Y 326.658,Z 165.275,A -85,B 0,C 180,E1 -15000.341,E2 -15000.341} C_VEL
LIN {X 0,Y 326.686,Z 165.294,A -85,B 0,C 180,E1 -15004.516,E2 -15004.516} C_VEL
LIN {X 0,Y 326.691,Z 165.587,A -85,B 0,C 180,E1 -15005.621,E2 -15005.621} C_VEL
LIN {X 0,Y 326.997,Z 166.824,A -85,B 0,C 180,E1 -15005.854,E2 -15005.854} C_VEL
LIN {X 0,Y 328.544,Z 169.353,A -85,B 0,C 180,E1 -15006.172,E2 -15006.172} C_VEL
LIN {X 0,Y 329.922,Z 170.862,A -85,B 0,C 180,E1 -15006.429,E2 -15006.429} C_VEL
LIN {X 0,Y 332.332,Z 174.357,A -85,B 0,C 180,E1 -15006.946,E2 -15006.946} C_VEL
LIN {X 0,Y 333.847,Z 176.146,A -85,B 0,C 180,E1 -15007.255,E2 -15007.255} C_VEL
LIN {X 0,Y 336.858,Z 179.834,A -85,B 0,C 180,E1 -15007.873,E2 -15007.873} C_VEL
LIN {X 0,Y 341.329,Z 185.197,A -85,B 0,C 180,E1 -15008.866,E2 -15008.866} C_VEL
LIN {X 0,Y 343.578,Z 187.673,A -85,B 0,C 180,E1 -15009.36,E2 -15009.36} C_VEL
LIN {X 0,Y 347.347,Z 191.645,A -85,B 0,C 180,E1 -15010.249,E2 -15010.249} C_VEL
LIN {X 0,Y 352.203,Z 196.917,A -85,B 0,C 180,E1 -15011.455,E2 -15011.455} C_VEL
LIN {X 0,Y 354.866,Z 199.388,A -85,B 0,C 180,E1 -15012.126,E2 -15012.126} C_VEL
LIN {X 0,Y 359.165,Z 203.614,A -85,B 0,C 180,E1 -15013.306,E2 -15013.306} C_VEL
LIN {X 0,Y 361.621,Z 205.668,A -85,B 0,C 180,E1 -15014.013,E2 -15014.013} C_VEL
LIN {X 0,Y 365.635,Z 209.686,A -85,B 0,C 180,E1 -15015.257,E2 -15015.257} C_VEL
LIN {X 0,Y 369.613,Z 212.872,A -85,B 0,C 180,E1 -15016.584,E2 -15016.584} C_VEL
LIN {X 0,Y 373.669,Z 216.74,A -85,B 0,C 180,E1 -15018.131,E2 -15018.131} C_VEL
LIN {X 0,Y 377.405,Z 219.212,A -85,B 0,C 180,E1 -15019.711,E2 -15019.711} C_VEL
LIN {X 0,Y 378.641,Z 220.158,A -85,B 0,C 180,E1 -15020.316,E2 -15020.316} C_VEL
LIN {X 0,Y 381.246,Z 222.96,A -85,B 0,C 180,E1 -15021.75,E2 -15021.75} C_VEL
LIN {X 0,Y 383.646,Z 224.871,A -85,B 0,C 180,E1 -15023.284,E2 -15023.284} C_VEL
LIN {X 0,Y 385.845,Z 226.138,A -85,B 0,C 180,E1 -15025.046,E2 -15025.046} C_VEL
LIN {X 0,Y 387.489,Z 226.713,A -85,B 0,C 180,E1 -15026.881,E2 -15026.881} C_VEL
LIN {X 0,Y 388.378,Z 227.295,A -85,B 0,C 180,E1 -15028.963,E2 -15028.963} C_VEL
LIN {X 0,Y 388.542,Z 227.227,A -85,B 0,C 180,E1 -15030,E2 -15030} C_VEL
LIN {X 0,Y 388.258,Z 227.183,A -85,B 0,C 180,E1 -15031.556,E2 -15031.556} C_VEL
LIN {X 0,Y 387.234,Z 226.669,A -85,B 0,C 180,E1 -15033.443,E2 -15033.443} C_VEL
LIN {X 0,Y 385.526,Z 225.999,A -85,B 0,C 180,E1 -15035.23,E2 -15035.23} C_VEL
LIN {X 0,Y 383.278,Z 224.592,A -85,B 0,C 180,E1 -15036.977,E2 -15036.977} C_VEL
LIN {X 0,Y 380.599,Z 222.31,A -85,B 0,C 180,E1 -15038.639,E2 -15038.639} C_VEL
LIN {X 0,Y 377.888,Z 219.451,A -85,B 0,C 180,E1 -15040.06,E2 -15040.06} C_VEL
LIN {X 0,Y 374.225,Z 217.199,A -85,B 0,C 180,E1 -15041.637,E2 -15041.637} C_VEL
LIN {X 0,Y 370.283,Z 213.606,A -85,B 0,C 180,E1 -15043.165,E2 -15043.165} C_VEL
LIN {X 0,Y 368.107,Z 211.584,A -85,B 0,C 180,E1 -15043.926,E2 -15043.926} C_VEL
LIN {X 0,Y 363.709,Z 207.954,A -85,B 0,C 180,E1 -15045.342,E2 -15045.342} C_VEL
LIN {X 0,Y 360.454,Z 204.596,A -85,B 0,C 180,E1 -15046.334,E2 -15046.334} C_VEL
LIN {X 0,Y 355.913,Z 200.562,A -85,B 0,C 180,E1 -15047.589,E2 -15047.589} C_VEL
LIN {X 0,Y 353.163,Z 197.706,A -85,B 0,C 180,E1 -15048.309,E2 -15048.309} C_VEL
LIN {X 0,Y 349.304,Z 193.886,A -85,B 0,C 180,E1 -15049.284,E2 -15049.284} C_VEL
LIN {X 0,Y 346.286,Z 190.674,A -85,B 0,C 180,E1 -15049.994,E2 -15049.994} C_VEL
LIN {X 0,Y 342.731,Z 186.542,A -85,B 0,C 180,E1 -15050.838,E2 -15050.838} C_VEL
LIN {X 0,Y 338.478,Z 181.938,A -85,B 0,C 180,E1 -15051.76,E2 -15051.76} C_VEL
LIN {X 0,Y 336.613,Z 179.601,A -85,B 0,C 180,E1 -15052.177,E2 -15052.177} C_VEL
LIN {X 0,Y 333.567,Z 175.716,A -85,B 0,C 180,E1 -15052.804,E2 -15052.804} C_VEL
LIN {X 0,Y 330.474,Z 171.844,A -85,B 0,C 180,E1 -15053.45,E2 -15053.45} C_VEL
LIN {X 0,Y 329.168,Z 169.925,A -85,B 0,C 180,E1 -15053.716,E2 -15053.716} C_VEL
LIN {X 0,Y 327.268,Z 167.481,A -85,B 0,C 180,E1 -15054.08,E2 -15054.08} C_VEL
LIN {X 0,Y 326.717,Z 165.742,A -85,B 0,C 180,E1 -15054.335,E2 -15054.335} C_VEL
LIN {X 0,Y 326.684,Z 165.294,A -85,B 0,C 180,E1 -15054.803,E2 -15054.803} C_VEL
LIN {X 0,Y 326.653,Z 165.281,A -85,B 0,C 180,E1 -15058.251,E2 -15058.251} C_VEL
LIN {X 0,Y 326.598,Z 165.299,A -85,B 0,C 180,E1 -15061.094,E2 -15061.094} C_VEL
LIN {X 0,Y 326.605,Z 165.273,A -85,B 0,C 180,E1 -15064.019,E2 -15064.019} C_VEL
LIN {X 0,Y 326.625,Z 165.297,A -85,B 0,C 180,E1 -15067.239,E2 -15067.239} C_VEL
LIN {X 0,Y 326.572,Z 165.261,A -85,B 0,C 180,E1 -15071.131,E2 -15071.131} C_VEL
LIN {X 0,Y 326.552,Z 165.293,A -85,B 0,C 180,E1 -15074.748,E2 -15074.748} C_VEL
LIN {X 0,Y 326.572,Z 165.299,A -85,B 0,C 180,E1 -15078.155,E2 -15078.155} C_VEL
LIN {X 0,Y 326.62,Z 165.299,A -85,B 0,C 180,E1 -15081.392,E2 -15081.392} C_VEL
LIN {X 0,Y 326.615,Z 165.281,A -85,B 0,C 180,E1 -15084.852,E2 -15084.852} C_VEL
LIN {X 0,Y 326.603,Z 165.298,A -85,B 0,C 180,E1 -15087.456,E2 -15087.456} C_VEL
LIN {X 0,Y 326.656,Z 165.29,A -85,B 0,C 180,E1 -15090.341,E2 -15090.341} C_VEL
LIN {X 0,Y 326.686,Z 165.28,A -85,B 0,C 180,E1 -15094.517,E2 -15094.517} C_VEL
LIN {X 0,Y 326.642,Z 165.287,A -85,B 0,C 180,E1 -15098.546,E2 -15098.546} C_VEL
LIN {X 0,Y 326.741,Z 165.253,A -85,B 0,C 180,E1 -15101.178,E2 -15101.178} C_VEL
LIN {X 0,Y 326.754,Z 165.282,A -85,B 0,C 180,E1 -15105.268,E2 -15105.268} C_VEL
LIN {X 0,Y 326.103,Z 165.363,A -85,B 0,C 180,E1 -15106.297,E2 -15106.297} C_VEL
LIN {X 0,Y 323.239,Z 165.705,A -85,B 0,C 180,E1 -15107.971,E2 -15107.971} C_VEL
LIN {X 0,Y 320.832,Z 165.991,A -85,B 0,C 180,E1 -15109.328,E2 -15109.328} C_VEL
LIN {X 0,Y 319.847,Z 166.11,A -85,B 0,C 180,E1 -15110.379,E2 -15110.379} C_VEL
LIN {X 0,Y 319.794,Z 166.118,A -85,B 0,C 180,E1 -15110.734,E2 -15110.734} C_VEL
LIN {X 0,Y 319.949,Z 166.127,A -85,B 0,C 180,E1 -15113.695,E2 -15113.695} C_VEL
LIN {X 0,Y 319.988,Z 166.111,A -85,B 0,C 180,E1 -15117.483,E2 -15117.483} C_VEL
LIN {X 0,Y 320.128,Z 166.073,A -85,B 0,C 180,E1 -15120.001,E2 -15120.001} C_VEL
LIN {X 0,Y 319.987,Z 166.117,A -85,B 0,C 180,E1 -15122.518,E2 -15122.518} C_VEL
LIN {X 0,Y 319.942,Z 166.126,A -85,B 0,C 180,E1 -15126.306,E2 -15126.306} C_VEL
LIN {X 0,Y 319.835,Z 166.113,A -85,B 0,C 180,E1 -15128.849,E2 -15128.849} C_VEL
LIN {X 0,Y 319.679,Z 166.155,A -85,B 0,C 180,E1 -15132.701,E2 -15132.701} C_VEL
LIN {X 0,Y 319.698,Z 166.157,A -85,B 0,C 180,E1 -15135.296,E2 -15135.296} C_VEL
LIN {X 0,Y 319.673,Z 166.134,A -85,B 0,C 180,E1 -15139.256,E2 -15139.256} C_VEL
LIN {X 0,Y 319.569,Z 166.176,A -85,B 0,C 180,E1 -15143.32,E2 -15143.32} C_VEL
LIN {X 0,Y 319.633,Z 166.148,A -85,B 0,C 180,E1 -15146.089,E2 -15146.089} C_VEL
LIN {X 0,Y 319.579,Z 166.166,A -85,B 0,C 180,E1 -15148.935,E2 -15148.935} C_VEL
LIN {X 0,Y 319.53,Z 166.18,A -85,B 0,C 180,E1 -15151.863,E2 -15151.863} C_VEL
LIN {X 0,Y 319.579,Z 166.167,A -85,B 0,C 180,E1 -15155.544,E2 -15155.544} C_VEL
LIN {X 0,Y 319.572,Z 166.177,A -85,B 0,C 180,E1 -15158.009,E2 -15158.009} C_VEL
LIN {X 0,Y 319.526,Z 166.18,A -85,B 0,C 180,E1 -15161.598,E2 -15161.598} C_VEL
LIN {X 0,Y 319.488,Z 166.182,A -85,B 0,C 180,E1 -15165.258,E2 -15165.258} C_VEL
LIN {X 0,Y 319.529,Z 166.162,A -85,B 0,C 180,E1 -15168.712,E2 -15168.712} C_VEL
LIN {X 0,Y 319.58,Z 166.18,A -85,B 0,C 180,E1 -15172.345,E2 -15172.345} C_VEL
LIN {X 0,Y 319.59,Z 166.289,A -85,B 0,C 180,E1 -15176.049,E2 -15176.049} C_VEL
LIN {X 0,Y 320.964,Z 172.754,A -85,B 0,C 180,E1 -15178.647,E2 -15178.647} C_VEL
LIN {X 0,Y 322.75,Z 181.936,A -85,B 0,C 180,E1 -15182.085,E2 -15182.085} C_VEL
LIN {X 0,Y 323.075,Z 186.232,A -85,B 0,C 180,E1 -15183.654,E2 -15183.654} C_VEL
LIN {X 0,Y 322.586,Z 189.926,A -85,B 0,C 180,E1 -15184.85,E2 -15184.85} C_VEL
LIN {X 0,Y 324.838,Z 200.086,A -85,B 0,C 180,E1 -15185.326,E2 -15185.326} C_VEL
LIN {X 0,Y 329.604,Z 224.903,A -85,B 0,C 180,E1 -15186.281,E2 -15186.281} C_VEL
LIN {X 0,Y 330.622,Z 232.075,A -85,B 0,C 180,E1 -15186.524,E2 -15186.524} C_VEL
LIN {X 0,Y 329.18,Z 295.973,A -85,B 0,C 180,E1 -15187.937,E2 -15187.937} C_VEL
LIN {X 0,Y 328.628,Z 306.284,A -85,B 0,C 180,E1 -15188.311,E2 -15188.311} C_VEL
LIN {X 0,Y 327.873,Z 315.796,A -85,B 0,C 180,E1 -15188.795,E2 -15188.795} C_VEL
LIN {X 0,Y 327.027,Z 324.869,A -85,B 0,C 180,E1 -15189.396,E2 -15189.396} C_VEL
LIN {X 0,Y 326.021,Z 334.001,A -85,B 0,C 180,E1 -15190.153,E2 -15190.153} C_VEL
LIN {X 0,Y 324.884,Z 342.995,A -85,B 0,C 180,E1 -15191.066,E2 -15191.066} C_VEL
LIN {X 0,Y 323.698,Z 351.721,A -85,B 0,C 180,E1 -15192.141,E2 -15192.141} C_VEL
LIN {X 0,Y 322.681,Z 359.115,A -85,B 0,C 180,E1 -15193.227,E2 -15193.227} C_VEL
LIN {X 0,Y 321.657,Z 366.643,A -85,B 0,C 180,E1 -15194.537,E2 -15194.537} C_VEL
LIN {X 0,Y 320.843,Z 372.539,A -85,B 0,C 180,E1 -15195.734,E2 -15195.734} C_VEL
LIN {X 0,Y 319.824,Z 379.074,A -85,B 0,C 180,E1 -15197.306,E2 -15197.306} C_VEL
LIN {X 0,Y 319.19,Z 383.575,A -85,B 0,C 180,E1 -15198.571,E2 -15198.571} C_VEL
LIN {X 0,Y 318.538,Z 389.069,A -85,B 0,C 180,E1 -15200.475,E2 -15200.475} C_VEL
LIN {X 0,Y 318.077,Z 393.394,A -85,B 0,C 180,E1 -15202.382,E2 -15202.382} C_VEL
LIN {X 0,Y 317.839,Z 396.666,A -85,B 0,C 180,E1 -15204.291,E2 -15204.291} C_VEL
LIN {X 0,Y 317.786,Z 398.952,A -85,B 0,C 180,E1 -15206.196,E2 -15206.196} C_VEL
LIN {X 0,Y 317.756,Z 400.011,A -85,B 0,C 180,E1 -15207.465,E2 -15207.465} C_VEL
LIN {X 0,Y 317.734,Z 400.599,A -85,B 0,C 180,E1 -15208.733,E2 -15208.733} C_VEL
LIN {X 0,Y 317.734,Z 400.599,A -85,B 0,C 180,E1 -15211.267,E2 -15211.267} C_VEL
LIN {X 0,Y 317.756,Z 400.011,A -85,B 0,C 180,E1 -15212.535,E2 -15212.535} C_VEL
LIN {X 0,Y 317.796,Z 397.562,A -85,B 0,C 180,E1 -15215.075,E2 -15215.075} C_VEL
LIN {X 0,Y 317.985,Z 394.612,A -85,B 0,C 180,E1 -15216.982,E2 -15216.982} C_VEL
LIN {X 0,Y 318.361,Z 390.623,A -85,B 0,C 180,E1 -15218.889,E2 -15218.889} C_VEL
LIN {X 0,Y 318.948,Z 385.492,A -85,B 0,C 180,E1 -15220.795,E2 -15220.795} C_VEL
LIN {X 0,Y 319.63,Z 380.229,A -85,B 0,C 180,E1 -15222.379,E2 -15222.379} C_VEL
LIN {X 0,Y 320.629,Z 373.914,A -85,B 0,C 180,E1 -15223.952,E2 -15223.952} C_VEL
LIN {X 0,Y 321.444,Z 367.962,A -85,B 0,C 180,E1 -15225.21,E2 -15225.21} C_VEL
LIN {X 0,Y 322.41,Z 361.034,A -85,B 0,C 180,E1 -15226.462,E2 -15226.462} C_VEL
LIN {X 0,Y 323.54,Z 352.855,A -85,B 0,C 180,E1 -15227.704,E2 -15227.704} C_VEL
LIN {X 0,Y 324.725,Z 344.346,A -85,B 0,C 180,E1 -15228.78,E2 -15228.78} C_VEL
LIN {X 0,Y 325.804,Z 335.632,A -85,B 0,C 180,E1 -15229.697,E2 -15229.697} C_VEL
LIN {X 0,Y 326.949,Z 325.877,A -85,B 0,C 180,E1 -15230.527,E2 -15230.527} C_VEL
LIN {X 0,Y 327.853,Z 315.796,A -85,B 0,C 180,E1 -15231.207,E2 -15231.207} C_VEL
LIN {X 0,Y 328.58,Z 306.283,A -85,B 0,C 180,E1 -15231.692,E2 -15231.692} C_VEL
LIN {X 0,Y 329.193,Z 295.974,A -85,B 0,C 180,E1 -15232.062,E2 -15232.062} C_VEL
LIN {X 0,Y 330.599,Z 231.386,A -85,B 0,C 180,E1 -15233.493,E2 -15233.493} C_VEL
LIN {X 0,Y 326.809,Z 209.434,A -85,B 0,C 180,E1 -15234.296,E2 -15234.296} C_VEL
LIN {X 0,Y 322.619,Z 190.102,A -85,B 0,C 180,E1 -15235.127,E2 -15235.127} C_VEL
LIN {X 0,Y 322.726,Z 188.615,A -85,B 0,C 180,E1 -15235.508,E2 -15235.508} C_VEL
LIN {X 0,Y 323.131,Z 184.669,A -85,B 0,C 180,E1 -15236.906,E2 -15236.906} C_VEL
LIN {X 0,Y 321.927,Z 177.478,A -85,B 0,C 180,E1 -15239.599,E2 -15239.599} C_VEL
LIN {X 0,Y 320.158,Z 168.873,A -85,B 0,C 180,E1 -15242.908,E2 -15242.908} C_VEL
LIN {X 0,Y 319.598,Z 166.189,A -85,B 0,C 180,E1 -15244.059,E2 -15244.059} C_VEL
LIN {X 0,Y 319.575,Z 166.177,A -85,B 0,C 180,E1 -15248.007,E2 -15248.007} C_VEL
LIN {X 0,Y 319.526,Z 166.166,A -85,B 0,C 180,E1 -15251.596,E2 -15251.596} C_VEL
LIN {X 0,Y 319.488,Z 166.18,A -85,B 0,C 180,E1 -15255.256,E2 -15255.256} C_VEL
LIN {X 0,Y 319.529,Z 166.179,A -85,B 0,C 180,E1 -15258.711,E2 -15258.711} C_VEL
LIN {X 0,Y 319.561,Z 166.178,A -85,B 0,C 180,E1 -15262.347,E2 -15262.347} C_VEL
LIN {X 0,Y 319.559,Z 166.161,A -85,B 0,C 180,E1 -15265.123,E2 -15265.123} C_VEL
LIN {X 0,Y 319.565,Z 166.18,A -85,B 0,C 180,E1 -15269.058,E2 -15269.058} C_VEL
LIN {X 0,Y 319.604,Z 166.15,A -85,B 0,C 180,E1 -15272.497,E2 -15272.497} C_VEL
LIN {X 0,Y 319.604,Z 166.165,A -85,B 0,C 180,E1 -15275.303,E2 -15275.303} C_VEL
LIN {X 0,Y 319.596,Z 166.17,A -85,B 0,C 180,E1 -15278.047,E2 -15278.047} C_VEL
LIN {X 0,Y 319.687,Z 166.131,A -85,B 0,C 180,E1 -15280.962,E2 -15280.962} C_VEL
LIN {X 0,Y 319.729,Z 166.155,A -85,B 0,C 180,E1 -15285.275,E2 -15285.275} C_VEL
LIN {X 0,Y 319.75,Z 166.121,A -85,B 0,C 180,E1 -15289.872,E2 -15289.872} C_VEL
LIN {X 0,Y 319.911,Z 166.117,A -85,B 0,C 180,E1 -15292.425,E2 -15292.425} C_VEL
LIN {X 0,Y 319.744,Z 166.156,A -85,B 0,C 180,E1 -15294.955,E2 -15294.955} C_VEL
LIN {X 0,Y 319.987,Z 166.117,A -85,B 0,C 180,E1 -15297.482,E2 -15297.482} C_VEL
LIN {X 0,Y 320.128,Z 166.073,A -85,B 0,C 180,E1 -15299.999,E2 -15299.999} C_VEL
LIN {X 0,Y 319.988,Z 166.111,A -85,B 0,C 180,E1 -15302.517,E2 -15302.517} C_VEL
LIN {X 0,Y 319.929,Z 166.125,A -85,B 0,C 180,E1 -15306.634,E2 -15306.634} C_VEL
LIN {X 0,Y 319.754,Z 166.121,A -85,B 0,C 180,E1 -15310.127,E2 -15310.127} C_VEL
LIN {X 0,Y 319.727,Z 166.157,A -85,B 0,C 180,E1 -15314.723,E2 -15314.723} C_VEL
LIN {X 0,Y 319.685,Z 166.131,A -85,B 0,C 180,E1 -15319.037,E2 -15319.037} C_VEL
LIN {X 0,Y 319.566,Z 166.178,A -85,B 0,C 180,E1 -15323.319,E2 -15323.319} C_VEL
LIN {X 0,Y 319.631,Z 166.152,A -85,B 0,C 180,E1 -15326.088,E2 -15326.088} C_VEL
LIN {X 0,Y 319.585,Z 166.164,A -85,B 0,C 180,E1 -15328.933,E2 -15328.933} C_VEL
LIN {X 0,Y 319.528,Z 166.182,A -85,B 0,C 180,E1 -15331.861,E2 -15331.861} C_VEL
LIN {X 0,Y 319.575,Z 166.162,A -85,B 0,C 180,E1 -15335.543,E2 -15335.543} C_VEL
LIN {X 0,Y 319.569,Z 166.178,A -85,B 0,C 180,E1 -15338.008,E2 -15338.008} C_VEL
LIN {X 0,Y 319.521,Z 166.173,A -85,B 0,C 180,E1 -15341.597,E2 -15341.597} C_VEL
LIN {X 0,Y 319.511,Z 166.177,A -85,B 0,C 180,E1 -15344.738,E2 -15344.738} C_VEL
LIN {X 0,Y 319.556,Z 166.133,A -85,B 0,C 180,E1 -15347.017,E2 -15347.017} C_VEL
LIN {X 0,Y 319.543,Z 166.165,A -85,B 0,C 180,E1 -15350.371,E2 -15350.371} C_VEL
LIN {X 0,Y 319.555,Z 166.167,A -85,B 0,C 180,E1 -15353.572,E2 -15353.572} C_VEL
LIN {X 0,Y 319.574,Z 166.156,A -85,B 0,C 180,E1 -15356.686,E2 -15356.686} C_VEL
LIN {X 0,Y 319.589,Z 166.161,A -85,B 0,C 180,E1 -15359.617,E2 -15359.617} C_VEL
LIN {X 0,Y 319.605,Z 166.171,A -85,B 0,C 180,E1 -15362.498,E2 -15362.498} C_VEL
LIN {X 0,Y 319.676,Z 166.392,A -85,B 0,C 180,E1 -15364.614,E2 -15364.614} C_VEL
LIN {X 0,Y 319.92,Z 167.459,A -85,B 0,C 180,E1 -15364.854,E2 -15364.854} C_VEL
LIN {X 0,Y 321.68,Z 170.339,A -85,B 0,C 180,E1 -15365.191,E2 -15365.191} C_VEL
LIN {X 0,Y 324.766,Z 174.853,A -85,B 0,C 180,E1 -15365.751,E2 -15365.751} C_VEL
LIN {X 0,Y 326.817,Z 177.585,A -85,B 0,C 180,E1 -15366.145,E2 -15366.145} C_VEL
LIN {X 0,Y 330.677,Z 182.38,A -85,B 0,C 180,E1 -15366.899,E2 -15366.899} C_VEL
LIN {X 0,Y 337.76,Z 190.702,A -85,B 0,C 180,E1 -15368.376,E2 -15368.376} C_VEL
LIN {X 0,Y 340.62,Z 193.804,A -85,B 0,C 180,E1 -15368.997,E2 -15368.997} C_VEL
LIN {X 0,Y 344.628,Z 197.86,A -85,B 0,C 180,E1 -15369.9,E2 -15369.9} C_VEL
LIN {X 0,Y 349.572,Z 203.113,A -85,B 0,C 180,E1 -15371.08,E2 -15371.08} C_VEL
LIN {X 0,Y 352.367,Z 205.723,A -85,B 0,C 180,E1 -15371.784,E2 -15371.784} C_VEL
LIN {X 0,Y 356.818,Z 209.996,A -85,B 0,C 180,E1 -15372.969,E2 -15372.969} C_VEL
LIN {X 0,Y 359.776,Z 212.469,A -85,B 0,C 180,E1 -15373.784,E2 -15373.784} C_VEL
LIN {X 0,Y 364,Z 216.513,A -85,B 0,C 180,E1 -15375.072,E2 -15375.072} C_VEL
LIN {X 0,Y 367.974,Z 219.699,A -85,B 0,C 180,E1 -15376.368,E2 -15376.368} C_VEL
LIN {X 0,Y 372.208,Z 223.577,A -85,B 0,C 180,E1 -15377.937,E2 -15377.937} C_VEL
LIN {X 0,Y 376.097,Z 226.103,A -85,B 0,C 180,E1 -15379.539,E2 -15379.539} C_VEL
LIN {X 0,Y 377.506,Z 227.245,A -85,B 0,C 180,E1 -15380.219,E2 -15380.219} C_VEL
LIN {X 0,Y 380.162,Z 229.986,A -85,B 0,C 180,E1 -15381.649,E2 -15381.649} C_VEL
LIN {X 0,Y 382.58,Z 231.841,A -85,B 0,C 180,E1 -15383.16,E2 -15383.16} C_VEL
LIN {X 0,Y 384.637,Z 233.029,A -85,B 0,C 180,E1 -15384.758,E2 -15384.758} C_VEL
LIN {X 0,Y 386.062,Z 233.613,A -85,B 0,C 180,E1 -15386.193,E2 -15386.193} C_VEL
LIN {X 0,Y 387.299,Z 234.162,A -85,B 0,C 180,E1 -15388.18,E2 -15388.18} C_VEL
LIN {X 0,Y 387.677,Z 234.273,A -85,B 0,C 180,E1 -15390,E2 -15390} C_VEL
LIN {X 0,Y 387.389,Z 234.231,A -85,B 0,C 180,E1 -15391.559,E2 -15391.559} C_VEL
LIN {X 0,Y 386.606,Z 233.79,A -85,B 0,C 180,E1 -15393.126,E2 -15393.126} C_VEL
LIN {X 0,Y 384.954,Z 233.189,A -85,B 0,C 180,E1 -15394.966,E2 -15394.966} C_VEL
LIN {X 0,Y 382.89,Z 232.034,A -85,B 0,C 180,E1 -15396.624,E2 -15396.624} C_VEL
LIN {X 0,Y 380.161,Z 229.997,A -85,B 0,C 180,E1 -15398.351,E2 -15398.351} C_VEL
LIN {X 0,Y 377.309,Z 227.034,A -85,B 0,C 180,E1 -15399.881,E2 -15399.881} C_VEL
LIN {X 0,Y 375.601,Z 225.829,A -85,B 0,C 180,E1 -15400.674,E2 -15400.674} C_VEL
LIN {X 0,Y 371.828,Z 223.307,A -85,B 0,C 180,E1 -15402.206,E2 -15402.206} C_VEL
LIN {X 0,Y 367.711,Z 219.468,A -85,B 0,C 180,E1 -15403.721,E2 -15403.721} C_VEL
LIN {X 0,Y 365.954,Z 217.984,A -85,B 0,C 180,E1 -15404.304,E2 -15404.304} C_VEL
LIN {X 0,Y 361.414,Z 214.229,A -85,B 0,C 180,E1 -15405.715,E2 -15405.715} C_VEL
LIN {X 0,Y 358.079,Z 210.927,A -85,B 0,C 180,E1 -15406.696,E2 -15406.696} C_VEL
LIN {X 0,Y 353.315,Z 206.717,A -85,B 0,C 180,E1 -15407.977,E2 -15407.977} C_VEL
LIN {X 0,Y 350.237,Z 203.678,A -85,B 0,C 180,E1 -15408.753,E2 -15408.753} C_VEL
LIN {X 0,Y 346.116,Z 199.577,A -85,B 0,C 180,E1 -15409.746,E2 -15409.746} C_VEL
LIN {X 0,Y 340.257,Z 193.367,A -85,B 0,C 180,E1 -15411.082,E2 -15411.082} C_VEL
LIN {X 0,Y 334.941,Z 187.429,A -85,B 0,C 180,E1 -15412.231,E2 -15412.231} C_VEL
LIN {X 0,Y 330.051,Z 181.459,A -85,B 0,C 180,E1 -15413.237,E2 -15413.237} C_VEL
LIN {X 0,Y 326.27,Z 176.733,A -85,B 0,C 180,E1 -15413.964,E2 -15413.964} C_VEL
LIN {X 0,Y 322.88,Z 172.255,A -85,B 0,C 180,E1 -15414.597,E2 -15414.597} C_VEL
LIN {X 0,Y 321.436,Z 170.076,A -85,B 0,C 180,E1 -15414.85,E2 -15414.85} C_VEL
LIN {X 0,Y 319.918,Z 167.407,A -85,B 0,C 180,E1 -15415.156,E2 -15415.156} C_VEL
LIN {X 0,Y 319.676,Z 166.396,A -85,B 0,C 180,E1 -15415.386,E2 -15415.386} C_VEL
LIN {X 0,Y 319.586,Z 166.155,A -85,B 0,C 180,E1 -15418.934,E2 -15418.934} C_VEL
LIN {X 0,Y 319.536,Z 166.184,A -85,B 0,C 180,E1 -15421.861,E2 -15421.861} C_VEL
LIN {X 0,Y 319.576,Z 166.15,A -85,B 0,C 180,E1 -15425.543,E2 -15425.543} C_VEL
LIN {X 0,Y 319.569,Z 166.179,A -85,B 0,C 180,E1 -15428.008,E2 -15428.008} C_VEL
LIN {X 0,Y 319.521,Z 166.134,A -85,B 0,C 180,E1 -15431.597,E2 -15431.597} C_VEL
LIN {X 0,Y 319.511,Z 166.17,A -85,B 0,C 180,E1 -15434.738,E2 -15434.738} C_VEL
LIN {X 0,Y 319.556,Z 166.179,A -85,B 0,C 180,E1 -15437.018,E2 -15437.018} C_VEL
LIN {X 0,Y 319.542,Z 166.17,A -85,B 0,C 180,E1 -15440.371,E2 -15440.371} C_VEL
LIN {X 0,Y 319.555,Z 166.176,A -85,B 0,C 180,E1 -15443.573,E2 -15443.573} C_VEL
LIN {X 0,Y 319.573,Z 166.163,A -85,B 0,C 180,E1 -15446.687,E2 -15446.687} C_VEL
LIN {X 0,Y 319.587,Z 166.175,A -85,B 0,C 180,E1 -15449.617,E2 -15449.617} C_VEL
LIN {X 0,Y 319.604,Z 166.149,A -85,B 0,C 180,E1 -15452.499,E2 -15452.499} C_VEL
LIN {X 0,Y 319.601,Z 166.169,A -85,B 0,C 180,E1 -15455.305,E2 -15455.305} C_VEL
LIN {X 0,Y 319.593,Z 166.17,A -85,B 0,C 180,E1 -15458.048,E2 -15458.048} C_VEL
LIN {X 0,Y 319.685,Z 166.131,A -85,B 0,C 180,E1 -15460.963,E2 -15460.963} C_VEL
LIN {X 0,Y 319.727,Z 166.157,A -85,B 0,C 180,E1 -15465.277,E2 -15465.277} C_VEL
LIN {X 0,Y 319.754,Z 166.121,A -85,B 0,C 180,E1 -15469.873,E2 -15469.873} C_VEL
LIN {X 0,Y 319.794,Z 166.118,A -85,B 0,C 180,E1 -15470.734,E2 -15470.734} C_VEL
LIN {X 0,Y 319.517,Z 166.159,A -85,B 0,C 180,E1 -15471.438,E2 -15471.438} C_VEL
LIN {X 0,Y 317.546,Z 166.421,A -85,B 0,C 180,E1 -15472.816,E2 -15472.816} C_VEL
LIN {X 0,Y 313.745,Z 166.906,A -85,B 0,C 180,E1 -15474.881,E2 -15474.881} C_VEL
LIN {X 0,Y 312.755,Z 167.024,A -85,B 0,C 180,E1 -15475.957,E2 -15475.957} C_VEL
LIN {X 0,Y 312.717,Z 167.024,A -85,B 0,C 180,E1 -15476.321,E2 -15476.321} C_VEL
LIN {X 0,Y 312.988,Z 166.969,A -85,B 0,C 180,E1 -15478.714,E2 -15478.714} C_VEL
LIN {X 0,Y 312.985,Z 166.972,A -85,B 0,C 180,E1 -15481.287,E2 -15481.287} C_VEL
LIN {X 0,Y 312.714,Z 167.033,A -85,B 0,C 180,E1 -15485.158,E2 -15485.158} C_VEL
LIN {X 0,Y 312.852,Z 166.994,A -85,B 0,C 180,E1 -15487.747,E2 -15487.747} C_VEL
LIN {X 0,Y 312.667,Z 167.018,A -85,B 0,C 180,E1 -15491.672,E2 -15491.672} C_VEL
LIN {X 0,Y 312.698,Z 167.032,A -85,B 0,C 180,E1 -15494.888,E2 -15494.888} C_VEL
LIN {X 0,Y 312.628,Z 167.01,A -85,B 0,C 180,E1 -15499.237,E2 -15499.237} C_VEL
LIN {X 0,Y 312.545,Z 167.051,A -85,B 0,C 180,E1 -15502.79,E2 -15502.79} C_VEL
LIN {X 0,Y 312.601,Z 167.025,A -85,B 0,C 180,E1 -15505.936,E2 -15505.936} C_VEL
LIN {X 0,Y 312.537,Z 167.051,A -85,B 0,C 180,E1 -15509.651,E2 -15509.651} C_VEL
LIN {X 0,Y 312.519,Z 167.036,A -85,B 0,C 180,E1 -15513.69,E2 -15513.69} C_VEL
LIN {X 0,Y 312.525,Z 167.055,A -85,B 0,C 180,E1 -15517.386,E2 -15517.386} C_VEL
LIN {X 0,Y 312.49,Z 167.048,A -85,B 0,C 180,E1 -15520.71,E2 -15520.71} C_VEL
LIN {X 0,Y 312.452,Z 167.057,A -85,B 0,C 180,E1 -15524.21,E2 -15524.21} C_VEL
LIN {X 0,Y 312.485,Z 167.05,A -85,B 0,C 180,E1 -15527.919,E2 -15527.919} C_VEL
LIN {X 0,Y 312.537,Z 167.053,A -85,B 0,C 180,E1 -15531.911,E2 -15531.911} C_VEL
LIN {X 0,Y 312.559,Z 167.188,A -85,B 0,C 180,E1 -15535.602,E2 -15535.602} C_VEL
LIN {X 0,Y 314.047,Z 174.248,A -85,B 0,C 180,E1 -15538.479,E2 -15538.479} C_VEL
LIN {X 0,Y 315.507,Z 181.729,A -85,B 0,C 180,E1 -15541.386,E2 -15541.386} C_VEL
LIN {X 0,Y 316.139,Z 186.474,A -85,B 0,C 180,E1 -15543.193,E2 -15543.193} C_VEL
LIN {X 0,Y 315.808,Z 189.605,A -85,B 0,C 180,E1 -15544.251,E2 -15544.251} C_VEL
LIN {X 0,Y 316.769,Z 194.193,A -85,B 0,C 180,E1 -15544.515,E2 -15544.515} C_VEL
LIN {X 0,Y 321.364,Z 216.05,A -85,B 0,C 180,E1 -15545.428,E2 -15545.428} C_VEL
LIN {X 0,Y 324.102,Z 232.126,A -85,B 0,C 180,E1 -15546.029,E2 -15546.029} C_VEL
LIN {X 0,Y 322.617,Z 295.782,A -85,B 0,C 180,E1 -15547.464,E2 -15547.464} C_VEL
LIN {X 0,Y 322.046,Z 306.093,A -85,B 0,C 180,E1 -15547.844,E2 -15547.844} C_VEL
LIN {X 0,Y 321.267,Z 315.605,A -85,B 0,C 180,E1 -15548.337,E2 -15548.337} C_VEL
LIN {X 0,Y 320.385,Z 324.677,A -85,B 0,C 180,E1 -15548.949,E2 -15548.949} C_VEL
LIN {X 0,Y 319.36,Z 333.809,A -85,B 0,C 180,E1 -15549.721,E2 -15549.721} C_VEL
LIN {X 0,Y 318.176,Z 342.803,A -85,B 0,C 180,E1 -15550.651,E2 -15550.651} C_VEL
LIN {X 0,Y 316.949,Z 351.529,A -85,B 0,C 180,E1 -15551.748,E2 -15551.748} C_VEL
LIN {X 0,Y 315.85,Z 358.922,A -85,B 0,C 180,E1 -15552.853,E2 -15552.853} C_VEL
LIN {X 0,Y 314.779,Z 366.62,A -85,B 0,C 180,E1 -15554.225,E2 -15554.225} C_VEL
LIN {X 0,Y 313.695,Z 373.722,A -85,B 0,C 180,E1 -15555.733,E2 -15555.733} C_VEL
LIN {X 0,Y 312.672,Z 380.036,A -85,B 0,C 180,E1 -15557.341,E2 -15557.341} C_VEL
LIN {X 0,Y 311.947,Z 385.299,A -85,B 0,C 180,E1 -15558.96,E2 -15558.96} C_VEL
LIN {X 0,Y 311.308,Z 390.43,A -85,B 0,C 180,E1 -15560.908,E2 -15560.908} C_VEL
LIN {X 0,Y 310.922,Z 394.42,A -85,B 0,C 180,E1 -15562.859,E2 -15562.859} C_VEL
LIN {X 0,Y 310.706,Z 397.37,A -85,B 0,C 180,E1 -15564.809,E2 -15564.809} C_VEL
LIN {X 0,Y 310.679,Z 399.819,A -85,B 0,C 180,E1 -15567.407,E2 -15567.407} C_VEL
LIN {X 0,Y 310.649,Z 400.408,A -85,B 0,C 180,E1 -15568.704,E2 -15568.704} C_VEL
LIN {X 0,Y 310.649,Z 400.408,A -85,B 0,C 180,E1 -15571.296,E2 -15571.296} C_VEL
LIN {X 0,Y 310.679,Z 399.819,A -85,B 0,C 180,E1 -15572.593,E2 -15572.593} C_VEL
LIN {X 0,Y 310.7,Z 397.37,A -85,B 0,C 180,E1 -15575.191,E2 -15575.191} C_VEL
LIN {X 0,Y 310.918,Z 394.42,A -85,B 0,C 180,E1 -15577.142,E2 -15577.142} C_VEL
LIN {X 0,Y 311.308,Z 390.43,A -85,B 0,C 180,E1 -15579.092,E2 -15579.092} C_VEL
LIN {X 0,Y 311.947,Z 385.299,A -85,B 0,C 180,E1 -15581.04,E2 -15581.04} C_VEL
LIN {X 0,Y 312.671,Z 380.036,A -85,B 0,C 180,E1 -15582.659,E2 -15582.659} C_VEL
LIN {X 0,Y 313.708,Z 373.722,A -85,B 0,C 180,E1 -15584.266,E2 -15584.266} C_VEL
LIN {X 0,Y 314.797,Z 366.574,A -85,B 0,C 180,E1 -15585.784,E2 -15585.784} C_VEL
LIN {X 0,Y 315.886,Z 358.923,A -85,B 0,C 180,E1 -15587.145,E2 -15587.145} C_VEL
LIN {X 0,Y 317.109,Z 350.395,A -85,B 0,C 180,E1 -15588.41,E2 -15588.41} C_VEL
LIN {X 0,Y 318.556,Z 340.1,A -85,B 0,C 180,E1 -15589.66,E2 -15589.66} C_VEL
LIN {X 0,Y 320.06,Z 327.698,A -85,B 0,C 180,E1 -15590.821,E2 -15590.821} C_VEL
LIN {X 0,Y 321.141,Z 316.892,A -85,B 0,C 180,E1 -15591.588,E2 -15591.588} C_VEL
LIN {X 0,Y 321.937,Z 306.965,A -85,B 0,C 180,E1 -15592.121,E2 -15592.121} C_VEL
LIN {X 0,Y 322.572,Z 297.114,A -85,B 0,C 180,E1 -15592.497,E2 -15592.497} C_VEL
LIN {X 0,Y 323.194,Z 272.97,A -85,B 0,C 180,E1 -15593.074,E2 -15593.074} C_VEL
LIN {X 0,Y 324.054,Z 231.415,A -85,B 0,C 180,E1 -15593.992,E2 -15593.992} C_VEL
LIN {X 0,Y 319.673,Z 207.364,A -85,B 0,C 180,E1 -15594.92,E2 -15594.92} C_VEL
LIN {X 0,Y 315.854,Z 189.963,A -85,B 0,C 180,E1 -15595.698,E2 -15595.698} C_VEL
LIN {X 0,Y 315.963,Z 188.515,A -85,B 0,C 180,E1 -15596.059,E2 -15596.059} C_VEL
LIN {X 0,Y 316.132,Z 185.361,A -85,B 0,C 180,E1 -15597.22,E2 -15597.22} C_VEL
LIN {X 0,Y 314.753,Z 177.766,A -85,B 0,C 180,E1 -15600.157,E2 -15600.157} C_VEL
LIN {X 0,Y 313.213,Z 170.181,A -85,B 0,C 180,E1 -15603.16,E2 -15603.16} C_VEL
LIN {X 0,Y 312.53,Z 167.077,A -85,B 0,C 180,E1 -15604.499,E2 -15604.499} C_VEL
LIN {X 0,Y 312.537,Z 167.053,A -85,B 0,C 180,E1 -15608.089,E2 -15608.089} C_VEL
LIN {X 0,Y 312.485,Z 167.049,A -85,B 0,C 180,E1 -15612.081,E2 -15612.081} C_VEL
LIN {X 0,Y 312.458,Z 167.059,A -85,B 0,C 180,E1 -15616.034,E2 -15616.034} C_VEL
LIN {X 0,Y 312.504,Z 167.044,A -85,B 0,C 180,E1 -15619.874,E2 -15619.874} C_VEL
LIN {X 0,Y 312.525,Z 167.055,A -85,B 0,C 180,E1 -15622.614,E2 -15622.614} C_VEL
LIN {X 0,Y 312.519,Z 167.036,A -85,B 0,C 180,E1 -15626.31,E2 -15626.31} C_VEL
LIN {X 0,Y 312.537,Z 167.051,A -85,B 0,C 180,E1 -15630.349,E2 -15630.349} C_VEL
LIN {X 0,Y 312.601,Z 167.025,A -85,B 0,C 180,E1 -15634.064,E2 -15634.064} C_VEL
LIN {X 0,Y 312.586,Z 167.044,A -85,B 0,C 180,E1 -15637.528,E2 -15637.528} C_VEL
LIN {X 0,Y 312.636,Z 167.009,A -85,B 0,C 180,E1 -15641.656,E2 -15641.656} C_VEL
LIN {X 0,Y 312.692,Z 167.031,A -85,B 0,C 180,E1 -15645.685,E2 -15645.685} C_VEL
LIN {X 0,Y 312.696,Z 167.001,A -85,B 0,C 180,E1 -15649.641,E2 -15649.641} C_VEL
LIN {X 0,Y 312.852,Z 166.994,A -85,B 0,C 180,E1 -15652.253,E2 -15652.253} C_VEL
LIN {X 0,Y 312.714,Z 167.033,A -85,B 0,C 180,E1 -15654.842,E2 -15654.842} C_VEL
LIN {X 0,Y 312.985,Z 166.972,A -85,B 0,C 180,E1 -15658.713,E2 -15658.713} C_VEL
LIN {X 0,Y 312.988,Z 166.969,A -85,B 0,C 180,E1 -15661.286,E2 -15661.286} C_VEL
LIN {X 0,Y 312.715,Z 167.03,A -85,B 0,C 180,E1 -15665.157,E2 -15665.157} C_VEL
LIN {X 0,Y 312.87,Z 166.996,A -85,B 0,C 180,E1 -15667.745,E2 -15667.745} C_VEL
LIN {X 0,Y 312.666,Z 167.018,A -85,B 0,C 180,E1 -15671.671,E2 -15671.671} C_VEL
LIN {X 0,Y 312.696,Z 167.033,A -85,B 0,C 180,E1 -15674.887,E2 -15674.887} C_VEL
LIN {X 0,Y 312.626,Z 167.01,A -85,B 0,C 180,E1 -15679.236,E2 -15679.236} C_VEL
LIN {X 0,Y 312.542,Z 167.052,A -85,B 0,C 180,E1 -15682.789,E2 -15682.789} C_VEL
LIN {X 0,Y 312.599,Z 167.029,A -85,B 0,C 180,E1 -15685.935,E2 -15685.935} C_VEL
LIN {X 0,Y 312.541,Z 167.047,A -85,B 0,C 180,E1 -15689.649,E2 -15689.649} C_VEL
LIN {X 0,Y 312.515,Z 167.037,A -85,B 0,C 180,E1 -15693.688,E2 -15693.688} C_VEL
LIN {X 0,Y 312.534,Z 167.057,A -85,B 0,C 180,E1 -15697.383,E2 -15697.383} C_VEL
LIN {X 0,Y 312.485,Z 167.044,A -85,B 0,C 180,E1 -15700.709,E2 -15700.709} C_VEL
LIN {X 0,Y 312.469,Z 167.06,A -85,B 0,C 180,E1 -15704.205,E2 -15704.205} C_VEL
LIN {X 0,Y 312.481,Z 167.009,A -85,B 0,C 180,E1 -15707.918,E2 -15707.918} C_VEL
LIN {X 0,Y 312.531,Z 167.056,A -85,B 0,C 180,E1 -15711.91,E2 -15711.91} C_VEL
LIN {X 0,Y 312.502,Z 167.027,A -85,B 0,C 180,E1 -15715.79,E2 -15715.79} C_VEL
LIN {X 0,Y 312.525,Z 167.052,A -85,B 0,C 180,E1 -15718.854,E2 -15718.854} C_VEL
LIN {X 0,Y 312.571,Z 167.035,A -85,B 0,C 180,E1 -15721.825,E2 -15721.825} C_VEL
LIN {X 0,Y 312.604,Z 167.217,A -85,B 0,C 180,E1 -15723.741,E2 -15723.741} C_VEL
LIN {X 0,Y 312.824,Z 168.1,A -85,B 0,C 180,E1 -15723.98,E2 -15723.98} C_VEL
LIN {X 0,Y 314.287,Z 170.862,A -85,B 0,C 180,E1 -15724.26,E2 -15724.26} C_VEL
LIN {X 0,Y 317.384,Z 175.455,A -85,B 0,C 180,E1 -15724.753,E2 -15724.753} C_VEL
LIN {X 0,Y 320.823,Z 180.318,A -85,B 0,C 180,E1 -15725.351,E2 -15725.351} C_VEL
LIN {X 0,Y 325.312,Z 185.815,A -85,B 0,C 180,E1 -15726.151,E2 -15726.151} C_VEL
LIN {X 0,Y 329.995,Z 191.322,A -85,B 0,C 180,E1 -15727.046,E2 -15727.046} C_VEL
LIN {X 0,Y 335.059,Z 197.054,A -85,B 0,C 180,E1 -15728.075,E2 -15728.075} C_VEL
LIN {X 0,Y 341.322,Z 203.557,A -85,B 0,C 180,E1 -15729.423,E2 -15729.423} C_VEL
LIN {X 0,Y 347.4,Z 209.744,A -85,B 0,C 180,E1 -15730.835,E2 -15730.835} C_VEL
LIN {X 0,Y 350.62,Z 212.829,A -85,B 0,C 180,E1 -15731.639,E2 -15731.639} C_VEL
LIN {X 0,Y 355.26,Z 216.957,A -85,B 0,C 180,E1 -15732.838,E2 -15732.838} C_VEL
LIN {X 0,Y 358.062,Z 219.482,A -85,B 0,C 180,E1 -15733.61,E2 -15733.61} C_VEL
LIN {X 0,Y 362.803,Z 223.694,A -85,B 0,C 180,E1 -15735.022,E2 -15735.022} C_VEL
LIN {X 0,Y 366.017,Z 226.208,A -85,B 0,C 180,E1 -15736.054,E2 -15736.054} C_VEL
LIN {X 0,Y 370.012,Z 229.855,A -85,B 0,C 180,E1 -15737.482,E2 -15737.482} C_VEL
LIN {X 0,Y 373.581,Z 232.358,A -85,B 0,C 180,E1 -15738.882,E2 -15738.882} C_VEL
LIN {X 0,Y 375.882,Z 233.802,A -85,B 0,C 180,E1 -15739.874,E2 -15739.874} C_VEL
LIN {X 0,Y 378.948,Z 236.876,A -85,B 0,C 180,E1 -15741.468,E2 -15741.468} C_VEL
LIN {X 0,Y 381.669,Z 238.906,A -85,B 0,C 180,E1 -15743.143,E2 -15743.143} C_VEL
LIN {X 0,Y 384.063,Z 240.238,A -85,B 0,C 180,E1 -15745.023,E2 -15745.023} C_VEL
LIN {X 0,Y 385.734,Z 240.807,A -85,B 0,C 180,E1 -15746.867,E2 -15746.867} C_VEL
LIN {X 0,Y 386.655,Z 241.383,A -85,B 0,C 180,E1 -15748.959,E2 -15748.959} C_VEL
LIN {X 0,Y 386.812,Z 241.32,A -85,B 0,C 180,E1 -15750,E2 -15750} C_VEL
LIN {X 0,Y 386.523,Z 241.254,A -85,B 0,C 180,E1 -15751.563,E2 -15751.563} C_VEL
LIN {X 0,Y 385.729,Z 240.835,A -85,B 0,C 180,E1 -15753.133,E2 -15753.133} C_VEL
LIN {X 0,Y 384.063,Z 240.239,A -85,B 0,C 180,E1 -15754.977,E2 -15754.977} C_VEL
LIN {X 0,Y 381.669,Z 238.911,A -85,B 0,C 180,E1 -15756.856,E2 -15756.856} C_VEL
LIN {X 0,Y 378.693,Z 236.648,A -85,B 0,C 180,E1 -15758.683,E2 -15758.683} C_VEL
LIN {X 0,Y 375.155,Z 233.179,A -85,B 0,C 180,E1 -15760.465,E2 -15760.465} C_VEL
LIN {X 0,Y 371.149,Z 230.691,A -85,B 0,C 180,E1 -15762.097,E2 -15762.097} C_VEL
LIN {X 0,Y 367.011,Z 227.186,A -85,B 0,C 180,E1 -15763.611,E2 -15763.611} C_VEL
LIN {X 0,Y 364.064,Z 224.613,A -85,B 0,C 180,E1 -15764.593,E2 -15764.593} C_VEL
LIN {X 0,Y 359.113,Z 220.498,A -85,B 0,C 180,E1 -15766.088,E2 -15766.088} C_VEL
LIN {X 0,Y 355.261,Z 216.943,A -85,B 0,C 180,E1 -15767.162,E2 -15767.162} C_VEL
LIN {X 0,Y 350.616,Z 212.844,A -85,B 0,C 180,E1 -15768.362,E2 -15768.362} C_VEL
LIN {X 0,Y 347.251,Z 209.57,A -85,B 0,C 180,E1 -15769.203,E2 -15769.203} C_VEL
LIN {X 0,Y 342.662,Z 204.954,A -85,B 0,C 180,E1 -15770.272,E2 -15770.272} C_VEL
LIN {X 0,Y 336.602,Z 198.697,A -85,B 0,C 180,E1 -15771.594,E2 -15771.594} C_VEL
LIN {X 0,Y 331.269,Z 192.894,A -85,B 0,C 180,E1 -15772.69,E2 -15772.69} C_VEL
LIN {X 0,Y 325.992,Z 186.607,A -85,B 0,C 180,E1 -15773.722,E2 -15773.722} C_VEL
LIN {X 0,Y 322.08,Z 181.84,A -85,B 0,C 180,E1 -15774.438,E2 -15774.438} C_VEL
LIN {X 0,Y 318.202,Z 176.747,A -85,B 0,C 180,E1 -15775.104,E2 -15775.104} C_VEL
LIN {X 0,Y 314.994,Z 171.911,A -85,B 0,C 180,E1 -15775.629,E2 -15775.629} C_VEL
LIN {X 0,Y 312.909,Z 168.386,A -85,B 0,C 180,E1 -15775.986,E2 -15775.986} C_VEL
LIN {X 0,Y 312.618,Z 167.334,A -85,B 0,C 180,E1 -15776.194,E2 -15776.194} C_VEL
LIN {X 0,Y 312.551,Z 167.054,A -85,B 0,C 180,E1 -15776.725,E2 -15776.725} C_VEL
LIN {X 0,Y 312.542,Z 167.032,A -85,B 0,C 180,E1 -15779.65,E2 -15779.65} C_VEL
LIN {X 0,Y 312.516,Z 167.029,A -85,B 0,C 180,E1 -15783.689,E2 -15783.689} C_VEL
LIN {X 0,Y 312.534,Z 167.054,A -85,B 0,C 180,E1 -15787.384,E2 -15787.384} C_VEL
LIN {X 0,Y 312.485,Z 167.019,A -85,B 0,C 180,E1 -15790.709,E2 -15790.709} C_VEL
LIN {X 0,Y 312.468,Z 167.037,A -85,B 0,C 180,E1 -15794.206,E2 -15794.206} C_VEL
LIN {X 0,Y 312.481,Z 167.056,A -85,B 0,C 180,E1 -15797.919,E2 -15797.919} C_VEL
LIN {X 0,Y 312.531,Z 167.055,A -85,B 0,C 180,E1 -15801.911,E2 -15801.911} C_VEL
LIN {X 0,Y 312.502,Z 167.036,A -85,B 0,C 180,E1 -15805.79,E2 -15805.79} C_VEL
LIN {X 0,Y 312.519,Z 167.057,A -85,B 0,C 180,E1 -15808.854,E2 -15808.854} C_VEL
LIN {X 0,Y 312.57,Z 167.029,A -85,B 0,C 180,E1 -15811.825,E2 -15811.825} C_VEL
LIN {X 0,Y 312.581,Z 167.039,A -85,B 0,C 180,E1 -15814.711,E2 -15814.711} C_VEL
LIN {X 0,Y 312.583,Z 167.047,A -85,B 0,C 180,E1 -15817.529,E2 -15817.529} C_VEL
LIN {X 0,Y 312.634,Z 167.011,A -85,B 0,C 180,E1 -15821.657,E2 -15821.657} C_VEL
LIN {X 0,Y 312.69,Z 167.036,A -85,B 0,C 180,E1 -15825.687,E2 -15825.687} C_VEL
LIN {X 0,Y 312.698,Z 167,A -85,B 0,C 180,E1 -15829.642,E2 -15829.642} C_VEL
LIN {X 0,Y 312.87,Z 166.996,A -85,B 0,C 180,E1 -15832.255,E2 -15832.255} C_VEL
LIN {X 0,Y 312.715,Z 167.03,A -85,B 0,C 180,E1 -15834.843,E2 -15834.843} C_VEL
LIN {X 0,Y 312.717,Z 167.024,A -85,B 0,C 180,E1 -15836.321,E2 -15836.321} C_VEL
LIN {X 0,Y 312.186,Z 167.084,A -85,B 0,C 180,E1 -15837.399,E2 -15837.399} C_VEL
LIN {X 0,Y 309.452,Z 167.405,A -85,B 0,C 180,E1 -15839.157,E2 -15839.157} C_VEL
LIN {X 0,Y 307.049,Z 167.705,A -85,B 0,C 180,E1 -15840.582,E2 -15840.582} C_VEL
LIN {X 0,Y 305.99,Z 167.846,A -85,B 0,C 180,E1 -15841.684,E2 -15841.684} C_VEL
LIN {X 0,Y 305.893,Z 167.862,A -85,B 0,C 180,E1 -15842.058,E2 -15842.058} C_VEL
LIN {X 0,Y 305.841,Z 167.882,A -85,B 0,C 180,E1 -15846.598,E2 -15846.598} C_VEL
LIN {X 0,Y 305.702,Z 167.869,A -85,B 0,C 180,E1 -15849.261,E2 -15849.261} C_VEL
LIN {X 0,Y 305.587,Z 167.915,A -85,B 0,C 180,E1 -15853.297,E2 -15853.297} C_VEL
LIN {X 0,Y 305.592,Z 167.909,A -85,B 0,C 180,E1 -15856.021,E2 -15856.021} C_VEL
LIN {X 0,Y 305.575,Z 167.89,A -85,B 0,C 180,E1 -15859.445,E2 -15859.445} C_VEL
LIN {X 0,Y 305.49,Z 167.932,A -85,B 0,C 180,E1 -15863.042,E2 -15863.042} C_VEL
LIN {X 0,Y 305.53,Z 167.902,A -85,B 0,C 180,E1 -15866.222,E2 -15866.222} C_VEL
LIN {X 0,Y 305.487,Z 167.922,A -85,B 0,C 180,E1 -15869.048,E2 -15869.048} C_VEL
LIN {X 0,Y 305.442,Z 167.935,A -85,B 0,C 180,E1 -15871.953,E2 -15871.953} C_VEL
LIN {X 0,Y 305.462,Z 167.919,A -85,B 0,C 180,E1 -15875.114,E2 -15875.114} C_VEL
LIN {X 0,Y 305.466,Z 167.929,A -85,B 0,C 180,E1 -15878.533,E2 -15878.533} C_VEL
LIN {X 0,Y 305.455,Z 167.938,A -85,B 0,C 180,E1 -15882.587,E2 -15882.587} C_VEL
LIN {X 0,Y 305.426,Z 167.942,A -85,B 0,C 180,E1 -15886.346,E2 -15886.346} C_VEL
LIN {X 0,Y 305.459,Z 167.906,A -85,B 0,C 180,E1 -15889.893,E2 -15889.893} C_VEL
LIN {X 0,Y 305.485,Z 167.919,A -85,B 0,C 180,E1 -15893.632,E2 -15893.632} C_VEL
LIN {X 0,Y 305.521,Z 168.067,A -85,B 0,C 180,E1 -15895.118,E2 -15895.118} C_VEL
LIN {X 0,Y 307.11,Z 175.565,A -85,B 0,C 180,E1 -15898.242,E2 -15898.242} C_VEL
LIN {X 0,Y 308.924,Z 185.042,A -85,B 0,C 180,E1 -15902.048,E2 -15902.048} C_VEL
LIN {X 0,Y 309.088,Z 188.838,A -85,B 0,C 180,E1 -15903.498,E2 -15903.498} C_VEL
LIN {X 0,Y 309.084,Z 189.773,A -85,B 0,C 180,E1 -15903.697,E2 -15903.697} C_VEL
LIN {X 0,Y 314.3,Z 213.945,A -85,B 0,C 180,E1 -15904.791,E2 -15904.791} C_VEL
LIN {X 0,Y 317.577,Z 232.582,A -85,B 0,C 180,E1 -15905.52,E2 -15905.52} C_VEL
LIN {X 0,Y 316.154,Z 294.314,A -85,B 0,C 180,E1 -15906.934,E2 -15906.934} C_VEL
LIN {X 0,Y 315.53,Z 305.027,A -85,B 0,C 180,E1 -15907.318,E2 -15907.318} C_VEL
LIN {X 0,Y 314.782,Z 314.125,A -85,B 0,C 180,E1 -15907.781,E2 -15907.781} C_VEL
LIN {X 0,Y 313.739,Z 324.485,A -85,B 0,C 180,E1 -15908.481,E2 -15908.481} C_VEL
LIN {X 0,Y 312.716,Z 333.618,A -85,B 0,C 180,E1 -15909.27,E2 -15909.27} C_VEL
LIN {X 0,Y 311.457,Z 342.61,A -85,B 0,C 180,E1 -15910.216,E2 -15910.216} C_VEL
LIN {X 0,Y 310.182,Z 351.337,A -85,B 0,C 180,E1 -15911.335,E2 -15911.335} C_VEL
LIN {X 0,Y 309.04,Z 358.73,A -85,B 0,C 180,E1 -15912.463,E2 -15912.463} C_VEL
LIN {X 0,Y 308.015,Z 365.96,A -85,B 0,C 180,E1 -15913.771,E2 -15913.771} C_VEL
LIN {X 0,Y 307.022,Z 372.153,A -85,B 0,C 180,E1 -15915.077,E2 -15915.077} C_VEL
LIN {X 0,Y 305.943,Z 378.689,A -85,B 0,C 180,E1 -15916.72,E2 -15916.72} C_VEL
LIN {X 0,Y 305.196,Z 383.19,A -85,B 0,C 180,E1 -15918.039,E2 -15918.039} C_VEL
LIN {X 0,Y 304.454,Z 388.683,A -85,B 0,C 180,E1 -15920.03,E2 -15920.03} C_VEL
LIN {X 0,Y 303.958,Z 393.01,A -85,B 0,C 180,E1 -15922.026,E2 -15922.026} C_VEL
LIN {X 0,Y 303.743,Z 395.378,A -85,B 0,C 180,E1 -15923.357,E2 -15923.357} C_VEL
LIN {X 0,Y 303.64,Z 397.179,A -85,B 0,C 180,E1 -15924.688,E2 -15924.688} C_VEL
LIN {X 0,Y 303.603,Z 399.628,A -85,B 0,C 180,E1 -15927.346,E2 -15927.346} C_VEL
LIN {X 0,Y 303.566,Z 400.217,A -85,B 0,C 180,E1 -15928.673,E2 -15928.673} C_VEL
LIN {X 0,Y 303.566,Z 400.217,A -85,B 0,C 180,E1 -15931.327,E2 -15931.327} C_VEL
LIN {X 0,Y 303.603,Z 399.628,A -85,B 0,C 180,E1 -15932.654,E2 -15932.654} C_VEL
LIN {X 0,Y 303.62,Z 397.178,A -85,B 0,C 180,E1 -15935.313,E2 -15935.313} C_VEL
LIN {X 0,Y 303.841,Z 394.227,A -85,B 0,C 180,E1 -15937.309,E2 -15937.309} C_VEL
LIN {X 0,Y 304.266,Z 390.238,A -85,B 0,C 180,E1 -15939.305,E2 -15939.305} C_VEL
LIN {X 0,Y 304.954,Z 385.107,A -85,B 0,C 180,E1 -15941.297,E2 -15941.297} C_VEL
LIN {X 0,Y 305.733,Z 379.844,A -85,B 0,C 180,E1 -15942.951,E2 -15942.951} C_VEL
LIN {X 0,Y 306.794,Z 373.529,A -85,B 0,C 180,E1 -15944.595,E2 -15944.595} C_VEL
LIN {X 0,Y 307.747,Z 367.578,A -85,B 0,C 180,E1 -15945.905,E2 -15945.905} C_VEL
LIN {X 0,Y 308.757,Z 360.649,A -85,B 0,C 180,E1 -15947.212,E2 -15947.212} C_VEL
LIN {X 0,Y 310.016,Z 352.471,A -85,B 0,C 180,E1 -15948.504,E2 -15948.504} C_VEL
LIN {X 0,Y 311.3,Z 343.963,A -85,B 0,C 180,E1 -15949.622,E2 -15949.622} C_VEL
LIN {X 0,Y 312.431,Z 335.247,A -85,B 0,C 180,E1 -15950.577,E2 -15950.577} C_VEL
LIN {X 0,Y 313.656,Z 325.493,A -85,B 0,C 180,E1 -15951.439,E2 -15951.439} C_VEL
LIN {X 0,Y 314.659,Z 315.413,A -85,B 0,C 180,E1 -15952.142,E2 -15952.142} C_VEL
LIN {X 0,Y 315.443,Z 305.9,A -85,B 0,C 180,E1 -15952.645,E2 -15952.645} C_VEL
LIN {X 0,Y 316.108,Z 295.591,A -85,B 0,C 180,E1 -15953.026,E2 -15953.026} C_VEL
LIN {X 0,Y 317.576,Z 232.86,A -85,B 0,C 180,E1 -15954.473,E2 -15954.473} C_VEL
LIN {X 0,Y 313.548,Z 209.985,A -85,B 0,C 180,E1 -15955.372,E2 -15955.372} C_VEL
LIN {X 0,Y 309.109,Z 189.745,A -85,B 0,C 180,E1 -15956.304,E2 -15956.304} C_VEL
LIN {X 0,Y 309.161,Z 188.32,A -85,B 0,C 180,E1 -15956.677,E2 -15956.677} C_VEL
LIN {X 0,Y 308.923,Z 185.041,A -85,B 0,C 180,E1 -15957.953,E2 -15957.953} C_VEL
LIN {X 0,Y 307.116,Z 175.565,A -85,B 0,C 180,E1 -15961.757,E2 -15961.757} C_VEL
LIN {X 0,Y 305.518,Z 167.958,A -85,B 0,C 180,E1 -15964.97,E2 -15964.97} C_VEL
LIN {X 0,Y 305.468,Z 167.923,A -85,B 0,C 180,E1 -15968.532,E2 -15968.532} C_VEL
LIN {X 0,Y 305.456,Z 167.934,A -85,B 0,C 180,E1 -15972.585,E2 -15972.585} C_VEL
LIN {X 0,Y 305.426,Z 167.937,A -85,B 0,C 180,E1 -15976.344,E2 -15976.344} C_VEL
LIN {X 0,Y 305.458,Z 167.922,A -85,B 0,C 180,E1 -15979.892,E2 -15979.892} C_VEL
LIN {X 0,Y 305.481,Z 167.928,A -85,B 0,C 180,E1 -15983.631,E2 -15983.631} C_VEL
LIN {X 0,Y 305.464,Z 167.915,A -85,B 0,C 180,E1 -15986.482,E2 -15986.482} C_VEL
LIN {X 0,Y 305.457,Z 167.935,A -85,B 0,C 180,E1 -15989.59,E2 -15989.59} C_VEL
LIN {X 0,Y 305.517,Z 167.902,A -85,B 0,C 180,E1 -15992.608,E2 -15992.608} C_VEL
LIN {X 0,Y 305.507,Z 167.924,A -85,B 0,C 180,E1 -15995.538,E2 -15995.538} C_VEL
LIN {X 0,Y 305.517,Z 167.906,A -85,B 0,C 180,E1 -15999.814,E2 -15999.814} C_VEL
LIN {X 0,Y 305.572,Z 167.895,A -85,B 0,C 180,E1 -16002.602,E2 -16002.602} C_VEL
LIN {X 0,Y 305.647,Z 167.909,A -85,B 0,C 180,E1 -16005.348,E2 -16005.348} C_VEL
LIN {X 0,Y 305.633,Z 167.882,A -85,B 0,C 180,E1 -16009.399,E2 -16009.399} C_VEL
LIN {X 0,Y 305.795,Z 167.872,A -85,B 0,C 180,E1 -16012.073,E2 -16012.073} C_VEL
LIN {X 0,Y 305.685,Z 167.909,A -85,B 0,C 180,E1 -16014.723,E2 -16014.723} C_VEL
LIN {X 0,Y 305.952,Z 167.847,A -85,B 0,C 180,E1 -16018.683,E2 -16018.683} C_VEL
LIN {X 0,Y 305.954,Z 167.844,A -85,B 0,C 180,E1 -16021.316,E2 -16021.316} C_VEL
LIN {X 0,Y 305.85,Z 167.88,A -85,B 0,C 180,E1 -16026.597,E2 -16026.597} C_VEL
LIN {X 0,Y 305.733,Z 167.868,A -85,B 0,C 180,E1 -16029.259,E2 -16029.259} C_VEL
LIN {X 0,Y 305.585,Z 167.915,A -85,B 0,C 180,E1 -16033.295,E2 -16033.295} C_VEL
LIN {X 0,Y 305.59,Z 167.913,A -85,B 0,C 180,E1 -16036.019,E2 -16036.019} C_VEL
LIN {X 0,Y 305.572,Z 167.888,A -85,B 0,C 180,E1 -16039.444,E2 -16039.444} C_VEL
LIN {X 0,Y 305.487,Z 167.931,A -85,B 0,C 180,E1 -16043.041,E2 -16043.041} C_VEL
LIN {X 0,Y 305.544,Z 167.905,A -85,B 0,C 180,E1 -16046.227,E2 -16046.227} C_VEL
LIN {X 0,Y 305.492,Z 167.92,A -85,B 0,C 180,E1 -16049.05,E2 -16049.05} C_VEL
LIN {X 0,Y 305.44,Z 167.936,A -85,B 0,C 180,E1 -16051.952,E2 -16051.952} C_VEL
LIN {X 0,Y 305.458,Z 167.915,A -85,B 0,C 180,E1 -16055.113,E2 -16055.113} C_VEL
LIN {X 0,Y 305.463,Z 167.935,A -85,B 0,C 180,E1 -16058.533,E2 -16058.533} C_VEL
LIN {X 0,Y 305.455,Z 167.934,A -85,B 0,C 180,E1 -16062.586,E2 -16062.586} C_VEL
LIN {X 0,Y 305.438,Z 167.899,A -85,B 0,C 180,E1 -16066.348,E2 -16066.348} C_VEL
LIN {X 0,Y 305.453,Z 167.905,A -85,B 0,C 180,E1 -16069.892,E2 -16069.892} C_VEL
LIN {X 0,Y 305.495,Z 167.915,A -85,B 0,C 180,E1 -16073.627,E2 -16073.627} C_VEL
LIN {X 0,Y 305.462,Z 167.909,A -85,B 0,C 180,E1 -16076.483,E2 -16076.483} C_VEL
LIN {X 0,Y 305.462,Z 167.919,A -85,B 0,C 180,E1 -16079.591,E2 -16079.591} C_VEL
LIN {X 0,Y 305.53,Z 168.083,A -85,B 0,C 180,E1 -16082.99,E2 -16082.99} C_VEL
LIN {X 0,Y 305.765,Z 169.097,A -85,B 0,C 180,E1 -16083.25,E2 -16083.25} C_VEL
LIN {X 0,Y 309.459,Z 175.536,A -85,B 0,C 180,E1 -16083.83,E2 -16083.83} C_VEL
LIN {X 0,Y 315.063,Z 183.694,A -85,B 0,C 180,E1 -16084.696,E2 -16084.696} C_VEL
LIN {X 0,Y 321.524,Z 191.39,A -85,B 0,C 180,E1 -16085.752,E2 -16085.752} C_VEL
LIN {X 0,Y 326.494,Z 197.078,A -85,B 0,C 180,E1 -16086.657,E2 -16086.657} C_VEL
LIN {X 0,Y 331.627,Z 202.791,A -85,B 0,C 180,E1 -16087.661,E2 -16087.661} C_VEL
LIN {X 0,Y 337.794,Z 209.183,A -85,B 0,C 180,E1 -16088.948,E2 -16088.948} C_VEL
LIN {X 0,Y 344.298,Z 215.637,A -85,B 0,C 180,E1 -16090.401,E2 -16090.401} C_VEL
LIN {X 0,Y 348.092,Z 219.121,A -85,B 0,C 180,E1 -16091.294,E2 -16091.294} C_VEL
LIN {X 0,Y 353.194,Z 223.548,A -85,B 0,C 180,E1 -16092.579,E2 -16092.579} C_VEL
LIN {X 0,Y 356.201,Z 226.257,A -85,B 0,C 180,E1 -16093.394,E2 -16093.394} C_VEL
LIN {X 0,Y 360.976,Z 230.382,A -85,B 0,C 180,E1 -16094.78,E2 -16094.78} C_VEL
LIN {X 0,Y 364.444,Z 233.12,A -85,B 0,C 180,E1 -16095.869,E2 -16095.869} C_VEL
LIN {X 0,Y 368.579,Z 236.72,A -85,B 0,C 180,E1 -16097.311,E2 -16097.311} C_VEL
LIN {X 0,Y 372.511,Z 239.385,A -85,B 0,C 180,E1 -16098.827,E2 -16098.827} C_VEL
LIN {X 0,Y 374.42,Z 240.551,A -85,B 0,C 180,E1 -16099.628,E2 -16099.628} C_VEL
LIN {X 0,Y 377.753,Z 243.768,A -85,B 0,C 180,E1 -16101.306,E2 -16101.306} C_VEL
LIN {X 0,Y 380.706,Z 245.935,A -85,B 0,C 180,E1 -16103.09,E2 -16103.09} C_VEL
LIN {X 0,Y 383.173,Z 247.283,A -85,B 0,C 180,E1 -16105.011,E2 -16105.011} C_VEL
LIN {X 0,Y 384.859,Z 247.83,A -85,B 0,C 180,E1 -16106.86,E2 -16106.86} C_VEL
LIN {X 0,Y 385.794,Z 248.43,A -85,B 0,C 180,E1 -16108.956,E2 -16108.956} C_VEL
LIN {X 0,Y 385.946,Z 248.367,A -85,B 0,C 180,E1 -16110,E2 -16110} C_VEL
LIN {X 0,Y 385.654,Z 248.302,A -85,B 0,C 180,E1 -16111.566,E2 -16111.566} C_VEL
LIN {X 0,Y 384.853,Z 247.87,A -85,B 0,C 180,E1 -16113.14,E2 -16113.14} C_VEL
LIN {X 0,Y 383.173,Z 247.284,A -85,B 0,C 180,E1 -16114.989,E2 -16114.989} C_VEL
LIN {X 0,Y 380.706,Z 245.935,A -85,B 0,C 180,E1 -16116.91,E2 -16116.91} C_VEL
LIN {X 0,Y 377.565,Z 243.647,A -85,B 0,C 180,E1 -16118.792,E2 -16118.792} C_VEL
LIN {X 0,Y 373.6,Z 239.945,A -85,B 0,C 180,E1 -16120.732,E2 -16120.732} C_VEL
LIN {X 0,Y 369.7,Z 237.566,A -85,B 0,C 180,E1 -16122.277,E2 -16122.277} C_VEL
LIN {X 0,Y 365.467,Z 234.1,A -85,B 0,C 180,E1 -16123.787,E2 -16123.787} C_VEL
LIN {X 0,Y 362.499,Z 231.442,A -85,B 0,C 180,E1 -16124.757,E2 -16124.757} C_VEL
LIN {X 0,Y 357.32,Z 227.381,A -85,B 0,C 180,E1 -16126.286,E2 -16126.286} C_VEL
LIN {X 0,Y 352.954,Z 223.364,A -85,B 0,C 180,E1 -16127.482,E2 -16127.482} C_VEL
LIN {X 0,Y 347.949,Z 219.006,A -85,B 0,C 180,E1 -16128.74,E2 -16128.74} C_VEL
LIN {X 0,Y 343.793,Z 215.171,A -85,B 0,C 180,E1 -16129.715,E2 -16129.715} C_VEL
LIN {X 0,Y 339.227,Z 210.452,A -85,B 0,C 180,E1 -16130.752,E2 -16130.752} C_VEL
LIN {X 0,Y 333.621,Z 204.855,A -85,B 0,C 180,E1 -16131.941,E2 -16131.941} C_VEL
LIN {X 0,Y 327.607,Z 198.432,A -85,B 0,C 180,E1 -16133.128,E2 -16133.128} C_VEL
LIN {X 0,Y 321.998,Z 191.931,A -85,B 0,C 180,E1 -16134.165,E2 -16134.165} C_VEL
LIN {X 0,Y 317.662,Z 186.763,A -85,B 0,C 180,E1 -16134.896,E2 -16134.896} C_VEL
LIN {X 0,Y 313.561,Z 181.591,A -85,B 0,C 180,E1 -16135.539,E2 -16135.539} C_VEL
LIN {X 0,Y 308.173,Z 173.646,A -85,B 0,C 180,E1 -16136.352,E2 -16136.352} C_VEL
LIN {X 0,Y 305.764,Z 169.104,A -85,B 0,C 180,E1 -16136.749,E2 -16136.749} C_VEL
LIN {X 0,Y 305.53,Z 168.086,A -85,B 0,C 180,E1 -16137.01,E2 -16137.01} C_VEL
LIN {X 0,Y 305.462,Z 167.919,A -85,B 0,C 180,E1 -16140.409,E2 -16140.409} C_VEL
LIN {X 0,Y 305.461,Z 167.904,A -85,B 0,C 180,E1 -16144.079,E2 -16144.079} C_VEL
LIN {X 0,Y 305.492,Z 167.923,A -85,B 0,C 180,E1 -16146.737,E2 -16146.737} C_VEL
LIN {X 0,Y 305.45,Z 167.896,A -85,B 0,C 180,E1 -16150.6,E2 -16150.6} C_VEL
LIN {X 0,Y 305.438,Z 167.899,A -85,B 0,C 180,E1 -16153.652,E2 -16153.652} C_VEL
LIN {X 0,Y 305.455,Z 167.934,A -85,B 0,C 180,E1 -16157.414,E2 -16157.414} C_VEL
LIN {X 0,Y 305.491,Z 167.931,A -85,B 0,C 180,E1 -16161.601,E2 -16161.601} C_VEL
LIN {X 0,Y 305.458,Z 167.915,A -85,B 0,C 180,E1 -16164.887,E2 -16164.887} C_VEL
LIN {X 0,Y 305.448,Z 167.937,A -85,B 0,C 180,E1 -16168.355,E2 -16168.355} C_VEL
LIN {X 0,Y 305.517,Z 167.916,A -85,B 0,C 180,E1 -16171.114,E2 -16171.114} C_VEL
LIN {X 0,Y 305.567,Z 167.904,A -85,B 0,C 180,E1 -16174.088,E2 -16174.088} C_VEL
LIN {X 0,Y 305.496,Z 167.922,A -85,B 0,C 180,E1 -16178.403,E2 -16178.403} C_VEL
LIN {X 0,Y 305.586,Z 167.886,A -85,B 0,C 180,E1 -16181.218,E2 -16181.218} C_VEL
LIN {X 0,Y 305.645,Z 167.912,A -85,B 0,C 180,E1 -16185.35,E2 -16185.35} C_VEL
LIN {X 0,Y 305.635,Z 167.881,A -85,B 0,C 180,E1 -16189.4,E2 -16189.4} C_VEL
LIN {X 0,Y 305.811,Z 167.871,A -85,B 0,C 180,E1 -16192.075,E2 -16192.075} C_VEL
LIN {X 0,Y 305.686,Z 167.906,A -85,B 0,C 180,E1 -16194.724,E2 -16194.724} C_VEL
LIN {X 0,Y 305.954,Z 167.844,A -85,B 0,C 180,E1 -16198.684,E2 -16198.684} C_VEL
LIN {X 0,Y 305.952,Z 167.847,A -85,B 0,C 180,E1 -16201.317,E2 -16201.317} C_VEL
LIN {X 0,Y 305.893,Z 167.862,A -85,B 0,C 180,E1 -16202.058,E2 -16202.058} C_VEL
LIN {X 0,Y 305.187,Z 167.963,A -85,B 0,C 180,E1 -16203.155,E2 -16203.155} C_VEL
LIN {X 0,Y 302.286,Z 168.331,A -85,B 0,C 180,E1 -16204.94,E2 -16204.94} C_VEL
LIN {X 0,Y 299.849,Z 168.628,A -85,B 0,C 180,E1 -16206.388,E2 -16206.388} C_VEL
LIN {X 0,Y 298.815,Z 168.744,A -85,B 0,C 180,E1 -16207.51,E2 -16207.51} C_VEL
LIN {X 0,Y 298.735,Z 168.749,A -85,B 0,C 180,E1 -16207.89,E2 -16207.89} C_VEL
LIN {X 0,Y 298.552,Z 168.785,A -85,B 0,C 180,E1 -16212.232,E2 -16212.232} C_VEL
LIN {X 0,Y 298.604,Z 168.785,A -85,B 0,C 180,E1 -16215.21,E2 -16215.21} C_VEL
LIN {X 0,Y 298.538,Z 168.764,A -85,B 0,C 180,E1 -16219.244,E2 -16219.244} C_VEL
LIN {X 0,Y 298.457,Z 168.804,A -85,B 0,C 180,E1 -16223.598,E2 -16223.598} C_VEL
LIN {X 0,Y 298.486,Z 168.777,A -85,B 0,C 180,E1 -16226.575,E2 -16226.575} C_VEL
LIN {X 0,Y 298.416,Z 168.811,A -85,B 0,C 180,E1 -16229.642,E2 -16229.642} C_VEL
LIN {X 0,Y 298.395,Z 168.801,A -85,B 0,C 180,E1 -16232.801,E2 -16232.801} C_VEL
LIN {X 0,Y 298.446,Z 168.809,A -85,B 0,C 180,E1 -16236.808,E2 -16236.808} C_VEL
LIN {X 0,Y 298.409,Z 168.801,A -85,B 0,C 180,E1 -16239.487,E2 -16239.487} C_VEL
LIN {X 0,Y 298.399,Z 168.813,A -85,B 0,C 180,E1 -16243.104,E2 -16243.104} C_VEL
LIN {X 0,Y 298.404,Z 168.815,A -85,B 0,C 180,E1 -16246.922,E2 -16246.922} C_VEL
LIN {X 0,Y 298.416,Z 168.792,A -85,B 0,C 180,E1 -16251.004,E2 -16251.004} C_VEL
LIN {X 0,Y 298.47,Z 168.874,A -85,B 0,C 180,E1 -16254.55,E2 -16254.55} C_VEL
LIN {X 0,Y 299.372,Z 173.284,A -85,B 0,C 180,E1 -16256.518,E2 -16256.518} C_VEL
LIN {X 0,Y 301.169,Z 182.193,A -85,B 0,C 180,E1 -16260.23,E2 -16260.23} C_VEL
LIN {X 0,Y 302.225,Z 188.642,A -85,B 0,C 180,E1 -16262.847,E2 -16262.847} C_VEL
LIN {X 0,Y 302.279,Z 189.542,A -85,B 0,C 180,E1 -16263.054,E2 -16263.054} C_VEL
LIN {X 0,Y 307.084,Z 211.025,A -85,B 0,C 180,E1 -16264.086,E2 -16264.086} C_VEL
LIN {X 0,Y 311.09,Z 233.283,A -85,B 0,C 180,E1 -16264.997,E2 -16264.997} C_VEL
LIN {X 0,Y 309.645,Z 294.129,A -85,B 0,C 180,E1 -16266.42,E2 -16266.42} C_VEL
LIN {X 0,Y 309.007,Z 304.836,A -85,B 0,C 180,E1 -16266.812,E2 -16266.812} C_VEL
LIN {X 0,Y 308.223,Z 313.934,A -85,B 0,C 180,E1 -16267.282,E2 -16267.282} C_VEL
LIN {X 0,Y 307.134,Z 324.293,A -85,B 0,C 180,E1 -16267.994,E2 -16267.994} C_VEL
LIN {X 0,Y 306.093,Z 333.427,A -85,B 0,C 180,E1 -16268.8,E2 -16268.8} C_VEL
LIN {X 0,Y 304.79,Z 342.419,A -85,B 0,C 180,E1 -16269.765,E2 -16269.765} C_VEL
LIN {X 0,Y 303.425,Z 351.144,A -85,B 0,C 180,E1 -16270.903,E2 -16270.903} C_VEL
LIN {X 0,Y 302.266,Z 358.538,A -85,B 0,C 180,E1 -16272.057,E2 -16272.057} C_VEL
LIN {X 0,Y 301.304,Z 364.813,A -85,B 0,C 180,E1 -16273.195,E2 -16273.195} C_VEL
LIN {X 0,Y 300.116,Z 371.96,A -85,B 0,C 180,E1 -16274.725,E2 -16274.725} C_VEL
LIN {X 0,Y 299.01,Z 378.497,A -85,B 0,C 180,E1 -16276.406,E2 -16276.406} C_VEL
LIN {X 0,Y 298.22,Z 382.997,A -85,B 0,C 180,E1 -16277.755,E2 -16277.755} C_VEL
LIN {X 0,Y 297.434,Z 388.491,A -85,B 0,C 180,E1 -16279.792,E2 -16279.792} C_VEL
LIN {X 0,Y 296.899,Z 392.817,A -85,B 0,C 180,E1 -16281.835,E2 -16281.835} C_VEL
LIN {X 0,Y 296.69,Z 395.186,A -85,B 0,C 180,E1 -16283.198,E2 -16283.198} C_VEL
LIN {X 0,Y 296.554,Z 396.987,A -85,B 0,C 180,E1 -16284.561,E2 -16284.561} C_VEL
LIN {X 0,Y 296.528,Z 399.437,A -85,B 0,C 180,E1 -16287.283,E2 -16287.283} C_VEL
LIN {X 0,Y 296.486,Z 400.026,A -85,B 0,C 180,E1 -16288.642,E2 -16288.642} C_VEL
LIN {X 0,Y 296.486,Z 400.026,A -85,B 0,C 180,E1 -16291.358,E2 -16291.358} C_VEL
LIN {X 0,Y 296.528,Z 399.437,A -85,B 0,C 180,E1 -16292.717,E2 -16292.717} C_VEL
LIN {X 0,Y 296.548,Z 396.895,A -85,B 0,C 180,E1 -16295.509,E2 -16295.509} C_VEL
LIN {X 0,Y 296.79,Z 394.035,A -85,B 0,C 180,E1 -16297.483,E2 -16297.483} C_VEL
LIN {X 0,Y 297.238,Z 390.045,A -85,B 0,C 180,E1 -16299.527,E2 -16299.527} C_VEL
LIN {X 0,Y 297.946,Z 384.914,A -85,B 0,C 180,E1 -16301.566,E2 -16301.566} C_VEL
LIN {X 0,Y 298.798,Z 379.652,A -85,B 0,C 180,E1 -16303.257,E2 -16303.257} C_VEL
LIN {X 0,Y 299.89,Z 373.337,A -85,B 0,C 180,E1 -16304.939,E2 -16304.939} C_VEL
LIN {X 0,Y 300.918,Z 367.387,A -85,B 0,C 180,E1 -16306.276,E2 -16306.276} C_VEL
LIN {X 0,Y 301.965,Z 360.457,A -85,B 0,C 180,E1 -16307.611,E2 -16307.611} C_VEL
LIN {X 0,Y 303.283,Z 352.279,A -85,B 0,C 180,E1 -16308.93,E2 -16308.93} C_VEL
LIN {X 0,Y 304.607,Z 343.771,A -85,B 0,C 180,E1 -16310.072,E2 -16310.072} C_VEL
LIN {X 0,Y 305.8,Z 335.056,A -85,B 0,C 180,E1 -16311.045,E2 -16311.045} C_VEL
LIN {X 0,Y 307.074,Z 325.301,A -85,B 0,C 180,E1 -16311.922,E2 -16311.922} C_VEL
LIN {X 0,Y 308.089,Z 315.221,A -85,B 0,C 180,E1 -16312.64,E2 -16312.64} C_VEL
LIN {X 0,Y 308.925,Z 305.709,A -85,B 0,C 180,E1 -16313.15,E2 -16313.15} C_VEL
LIN {X 0,Y 309.594,Z 295.4,A -85,B 0,C 180,E1 -16313.54,E2 -16313.54} C_VEL
LIN {X 0,Y 311.117,Z 233.735,A -85,B 0,C 180,E1 -16314.989,E2 -16314.989} C_VEL
LIN {X 0,Y 307.084,Z 211.018,A -85,B 0,C 180,E1 -16315.914,E2 -16315.914} C_VEL
LIN {X 0,Y 302.295,Z 189.526,A -85,B 0,C 180,E1 -16316.946,E2 -16316.946} C_VEL
LIN {X 0,Y 302.195,Z 188.119,A -85,B 0,C 180,E1 -16317.343,E2 -16317.343} C_VEL
LIN {X 0,Y 300.961,Z 181.075,A -85,B 0,C 180,E1 -16320.228,E2 -16320.228} C_VEL
LIN {X 0,Y 299.405,Z 173.328,A -85,B 0,C 180,E1 -16323.478,E2 -16323.478} C_VEL
LIN {X 0,Y 298.47,Z 168.874,A -85,B 0,C 180,E1 -16325.452,E2 -16325.452} C_VEL
LIN {X 0,Y 298.41,Z 168.787,A -85,B 0,C 180,E1 -16329.486,E2 -16329.486} C_VEL
LIN {X 0,Y 298.4,Z 168.815,A -85,B 0,C 180,E1 -16333.103,E2 -16333.103} C_VEL
LIN {X 0,Y 298.404,Z 168.814,A -85,B 0,C 180,E1 -16336.92,E2 -16336.92} C_VEL
LIN {X 0,Y 298.415,Z 168.803,A -85,B 0,C 180,E1 -16341.003,E2 -16341.003} C_VEL
LIN {X 0,Y 298.419,Z 168.806,A -85,B 0,C 180,E1 -16343.929,E2 -16343.929} C_VEL
LIN {X 0,Y 298.393,Z 168.813,A -85,B 0,C 180,E1 -16347.983,E2 -16347.983} C_VEL
LIN {X 0,Y 298.458,Z 168.788,A -85,B 0,C 180,E1 -16351.903,E2 -16351.903} C_VEL
LIN {X 0,Y 298.484,Z 168.79,A -85,B 0,C 180,E1 -16354.923,E2 -16354.923} C_VEL
LIN {X 0,Y 298.448,Z 168.792,A -85,B 0,C 180,E1 -16359.314,E2 -16359.314} C_VEL
LIN {X 0,Y 298.536,Z 168.767,A -85,B 0,C 180,E1 -16362.179,E2 -16362.179} C_VEL
LIN {X 0,Y 298.592,Z 168.789,A -85,B 0,C 180,E1 -16364.994,E2 -16364.994} C_VEL
LIN {X 0,Y 298.589,Z 168.761,A -85,B 0,C 180,E1 -16369.146,E2 -16369.146} C_VEL
LIN {X 0,Y 298.739,Z 168.747,A -85,B 0,C 180,E1 -16371.885,E2 -16371.885} C_VEL
LIN {X 0,Y 298.655,Z 168.783,A -85,B 0,C 180,E1 -16374.598,E2 -16374.598} C_VEL
LIN {X 0,Y 298.919,Z 168.723,A -85,B 0,C 180,E1 -16378.652,E2 -16378.652} C_VEL
LIN {X 0,Y 298.921,Z 168.719,A -85,B 0,C 180,E1 -16381.346,E2 -16381.346} C_VEL
LIN {X 0,Y 298.795,Z 168.758,A -85,B 0,C 180,E1 -16386.753,E2 -16386.753} C_VEL
LIN {X 0,Y 298.677,Z 168.744,A -85,B 0,C 180,E1 -16389.48,E2 -16389.48} C_VEL
LIN {X 0,Y 298.548,Z 168.793,A -85,B 0,C 180,E1 -16393.615,E2 -16393.615} C_VEL
LIN {X 0,Y 298.545,Z 168.788,A -85,B 0,C 180,E1 -16396.408,E2 -16396.408} C_VEL
LIN {X 0,Y 298.507,Z 168.769,A -85,B 0,C 180,E1 -16399.654,E2 -16399.654} C_VEL
LIN {X 0,Y 298.454,Z 168.81,A -85,B 0,C 180,E1 -16403.597,E2 -16403.597} C_VEL
LIN {X 0,Y 298.486,Z 168.78,A -85,B 0,C 180,E1 -16406.574,E2 -16406.574} C_VEL
LIN {X 0,Y 298.417,Z 168.806,A -85,B 0,C 180,E1 -16409.64,E2 -16409.64} C_VEL
LIN {X 0,Y 298.391,Z 168.808,A -85,B 0,C 180,E1 -16412.8,E2 -16412.8} C_VEL
LIN {X 0,Y 298.46,Z 168.805,A -85,B 0,C 180,E1 -16416.812,E2 -16416.812} C_VEL
LIN {X 0,Y 298.383,Z 168.801,A -85,B 0,C 180,E1 -16421.087,E2 -16421.087} C_VEL
LIN {X 0,Y 298.384,Z 168.803,A -85,B 0,C 180,E1 -16425.041,E2 -16425.041} C_VEL
LIN {X 0,Y 298.382,Z 168.768,A -85,B 0,C 180,E1 -16428.912,E2 -16428.912} C_VEL
LIN {X 0,Y 298.46,Z 168.8,A -85,B 0,C 180,E1 -16433.188,E2 -16433.188} C_VEL
LIN {X 0,Y 298.394,Z 168.801,A -85,B 0,C 180,E1 -16437.2,E2 -16437.2} C_VEL
LIN {X 0,Y 298.428,Z 168.788,A -85,B 0,C 180,E1 -16440.614,E2 -16440.614} C_VEL
LIN {X 0,Y 298.522,Z 169.066,A -85,B 0,C 180,E1 -16442.381,E2 -16442.381} C_VEL
LIN {X 0,Y 298.789,Z 170.11,A -85,B 0,C 180,E1 -16442.597,E2 -16442.597} C_VEL
LIN {X 0,Y 303.704,Z 179.102,A -85,B 0,C 180,E1 -16443.333,E2 -16443.333} C_VEL
LIN {X 0,Y 310.878,Z 189.154,A -85,B 0,C 180,E1 -16444.348,E2 -16444.348} C_VEL
LIN {X 0,Y 317.261,Z 196.573,A -85,B 0,C 180,E1 -16445.325,E2 -16445.325} C_VEL
LIN {X 0,Y 322.931,Z 202.826,A -85,B 0,C 180,E1 -16446.276,E2 -16446.276} C_VEL
LIN {X 0,Y 328.372,Z 208.716,A -85,B 0,C 180,E1 -16447.287,E2 -16447.287} C_VEL
LIN {X 0,Y 335.007,Z 215.431,A -85,B 0,C 180,E1 -16448.625,E2 -16448.625} C_VEL
LIN {X 0,Y 341.638,Z 221.904,A -85,B 0,C 180,E1 -16450.065,E2 -16450.065} C_VEL
LIN {X 0,Y 348.9,Z 228.462,A -85,B 0,C 180,E1 -16451.784,E2 -16451.784} C_VEL
LIN {X 0,Y 353.427,Z 232.21,A -85,B 0,C 180,E1 -16452.936,E2 -16452.936} C_VEL
LIN {X 0,Y 358.496,Z 236.566,A -85,B 0,C 180,E1 -16454.352,E2 -16454.352} C_VEL
LIN {X 0,Y 362.861,Z 240.008,A -85,B 0,C 180,E1 -16455.68,E2 -16455.68} C_VEL
LIN {X 0,Y 367.471,Z 243.838,A -85,B 0,C 180,E1 -16457.26,E2 -16457.26} C_VEL
LIN {X 0,Y 371.534,Z 246.453,A -85,B 0,C 180,E1 -16458.809,E2 -16458.809} C_VEL
LIN {X 0,Y 373.558,Z 247.937,A -85,B 0,C 180,E1 -16459.672,E2 -16459.672} C_VEL
LIN {X 0,Y 377.053,Z 251.109,A -85,B 0,C 180,E1 -16461.424,E2 -16461.424} C_VEL
LIN {X 0,Y 380.082,Z 253.162,A -85,B 0,C 180,E1 -16463.274,E2 -16463.274} C_VEL
LIN {X 0,Y 382.594,Z 254.44,A -85,B 0,C 180,E1 -16465.263,E2 -16465.263} C_VEL
LIN {X 0,Y 384.297,Z 255.053,A -85,B 0,C 180,E1 -16467.367,E2 -16467.367} C_VEL
LIN {X 0,Y 384.932,Z 255.473,A -85,B 0,C 180,E1 -16468.954,E2 -16468.954} C_VEL
LIN {X 0,Y 385.081,Z 255.414,A -85,B 0,C 180,E1 -16470,E2 -16470} C_VEL
LIN {X 0,Y 384.785,Z 255.35,A -85,B 0,C 180,E1 -16471.57,E2 -16471.57} C_VEL
LIN {X 0,Y 383.978,Z 254.898,A -85,B 0,C 180,E1 -16473.148,E2 -16473.148} C_VEL
LIN {X 0,Y 382.282,Z 254.33,A -85,B 0,C 180,E1 -16475.001,E2 -16475.001} C_VEL
LIN {X 0,Y 379.791,Z 252.994,A -85,B 0,C 180,E1 -16476.927,E2 -16476.927} C_VEL
LIN {X 0,Y 376.552,Z 250.734,A -85,B 0,C 180,E1 -16478.839,E2 -16478.839} C_VEL
LIN {X 0,Y 372.964,Z 247.385,A -85,B 0,C 180,E1 -16480.594,E2 -16480.594} C_VEL
LIN {X 0,Y 368.428,Z 244.567,A -85,B 0,C 180,E1 -16482.386,E2 -16482.386} C_VEL
LIN {X 0,Y 363.9,Z 241.004,A -85,B 0,C 180,E1 -16483.968,E2 -16483.968} C_VEL
LIN {X 0,Y 360.414,Z 237.989,A -85,B 0,C 180,E1 -16485.081,E2 -16485.081} C_VEL
LIN {X 0,Y 354.989,Z 233.735,A -85,B 0,C 180,E1 -16486.632,E2 -16486.632} C_VEL
LIN {X 0,Y 350.683,Z 229.833,A -85,B 0,C 180,E1 -16487.781,E2 -16487.781} C_VEL
LIN {X 0,Y 345.17,Z 225.104,A -85,B 0,C 180,E1 -16489.127,E2 -16489.127} C_VEL
LIN {X 0,Y 338.009,Z 218.527,A -85,B 0,C 180,E1 -16490.729,E2 -16490.729} C_VEL
LIN {X 0,Y 330.061,Z 210.475,A -85,B 0,C 180,E1 -16492.378,E2 -16492.378} C_VEL
LIN {X 0,Y 323.726,Z 203.789,A -85,B 0,C 180,E1 -16493.574,E2 -16493.574} C_VEL
LIN {X 0,Y 317.501,Z 196.819,A -85,B 0,C 180,E1 -16494.637,E2 -16494.637} C_VEL
LIN {X 0,Y 312.994,Z 191.53,A -85,B 0,C 180,E1 -16495.34,E2 -16495.34} C_VEL
LIN {X 0,Y 308.933,Z 186.551,A -85,B 0,C 180,E1 -16495.935,E2 -16495.935} C_VEL
LIN {X 0,Y 302.671,Z 177.407,A -85,B 0,C 180,E1 -16496.811,E2 -16496.811} C_VEL
LIN {X 0,Y 298.715,Z 169.91,A -85,B 0,C 180,E1 -16497.429,E2 -16497.429} C_VEL
LIN {X 0,Y 298.49,Z 168.901,A -85,B 0,C 180,E1 -16497.727,E2 -16497.727} C_VEL
LIN {X 0,Y 298.396,Z 168.817,A -85,B 0,C 180,E1 -16502.018,E2 -16502.018} C_VEL
LIN {X 0,Y 298.427,Z 168.789,A -85,B 0,C 180,E1 -16506.068,E2 -16506.068} C_VEL
LIN {X 0,Y 298.404,Z 168.797,A -85,B 0,C 180,E1 -16509.486,E2 -16509.486} C_VEL
LIN {X 0,Y 298.394,Z 168.767,A -85,B 0,C 180,E1 -16513.104,E2 -16513.104} C_VEL
LIN {X 0,Y 298.398,Z 168.816,A -85,B 0,C 180,E1 -16516.921,E2 -16516.921} C_VEL
LIN {X 0,Y 298.411,Z 168.809,A -85,B 0,C 180,E1 -16521.004,E2 -16521.004} C_VEL
LIN {X 0,Y 298.427,Z 168.802,A -85,B 0,C 180,E1 -16523.932,E2 -16523.932} C_VEL
LIN {X 0,Y 298.391,Z 168.813,A -85,B 0,C 180,E1 -16527.984,E2 -16527.984} C_VEL
LIN {X 0,Y 298.459,Z 168.784,A -85,B 0,C 180,E1 -16531.905,E2 -16531.905} C_VEL
LIN {X 0,Y 298.482,Z 168.798,A -85,B 0,C 180,E1 -16534.925,E2 -16534.925} C_VEL
LIN {X 0,Y 298.446,Z 168.789,A -85,B 0,C 180,E1 -16539.316,E2 -16539.316} C_VEL
LIN {X 0,Y 298.534,Z 168.771,A -85,B 0,C 180,E1 -16542.18,E2 -16542.18} C_VEL
LIN {X 0,Y 298.59,Z 168.79,A -85,B 0,C 180,E1 -16544.995,E2 -16544.995} C_VEL
LIN {X 0,Y 298.59,Z 168.76,A -85,B 0,C 180,E1 -16549.147,E2 -16549.147} C_VEL
LIN {X 0,Y 298.757,Z 168.747,A -85,B 0,C 180,E1 -16551.887,E2 -16551.887} C_VEL
LIN {X 0,Y 298.657,Z 168.781,A -85,B 0,C 180,E1 -16554.6,E2 -16554.6} C_VEL
LIN {X 0,Y 298.921,Z 168.719,A -85,B 0,C 180,E1 -16558.654,E2 -16558.654} C_VEL
LIN {X 0,Y 298.919,Z 168.723,A -85,B 0,C 180,E1 -16561.348,E2 -16561.348} C_VEL
LIN {X 0,Y 298.786,Z 168.758,A -85,B 0,C 180,E1 -16566.755,E2 -16566.755} C_VEL
LIN {X 0,Y 298.735,Z 168.749,A -85,B 0,C 180,E1 -16567.89,E2 -16567.89} C_VEL
LIN {X 0,Y 298.052,Z 168.829,A -85,B 0,C 180,E1 -16569.014,E2 -16569.014} C_VEL
LIN {X 0,Y 295.098,Z 169.199,A -85,B 0,C 180,E1 -16570.841,E2 -16570.841} C_VEL
LIN {X 0,Y 292.611,Z 169.525,A -85,B 0,C 180,E1 -16572.323,E2 -16572.323} C_VEL
LIN {X 0,Y 291.58,Z 169.661,A -85,B 0,C 180,E1 -16573.474,E2 -16573.474} C_VEL
LIN {X 0,Y 291.515,Z 169.668,A -85,B 0,C 180,E1 -16573.865,E2 -16573.865} C_VEL
LIN {X 0,Y 291.485,Z 169.655,A -85,B 0,C 180,E1 -16576.819,E2 -16576.819} C_VEL
LIN {X 0,Y 291.45,Z 169.652,A -85,B 0,C 180,E1 -16579.876,E2 -16579.876} C_VEL
LIN {X 0,Y 291.4,Z 169.683,A -85,B 0,C 180,E1 -16584.206,E2 -16584.206} C_VEL
LIN {X 0,Y 291.419,Z 169.656,A -85,B 0,C 180,E1 -16587.273,E2 -16587.273} C_VEL
LIN {X 0,Y 291.334,Z 169.695,A -85,B 0,C 180,E1 -16590.438,E2 -16590.438} C_VEL
LIN {X 0,Y 291.344,Z 169.672,A -85,B 0,C 180,E1 -16593.699,E2 -16593.699} C_VEL
LIN {X 0,Y 291.381,Z 169.689,A -85,B 0,C 180,E1 -16597.256,E2 -16597.256} C_VEL
LIN {X 0,Y 291.334,Z 169.681,A -85,B 0,C 180,E1 -16600.643,E2 -16600.643} C_VEL
LIN {X 0,Y 291.291,Z 169.691,A -85,B 0,C 180,E1 -16604.403,E2 -16604.403} C_VEL
LIN {X 0,Y 291.327,Z 169.675,A -85,B 0,C 180,E1 -16608.405,E2 -16608.405} C_VEL
LIN {X 0,Y 291.366,Z 169.672,A -85,B 0,C 180,E1 -16611.161,E2 -16611.161} C_VEL
LIN {X 0,Y 291.438,Z 169.863,A -85,B 0,C 180,E1 -16614.106,E2 -16614.106} C_VEL
LIN {X 0,Y 293.108,Z 177.886,A -85,B 0,C 180,E1 -16617.664,E2 -16617.664} C_VEL
LIN {X 0,Y 294.847,Z 186.954,A -85,B 0,C 180,E1 -16621.529,E2 -16621.529} C_VEL
LIN {X 0,Y 295.26,Z 189.127,A -85,B 0,C 180,E1 -16622.332,E2 -16622.332} C_VEL
LIN {X 0,Y 296.808,Z 194.647,A -85,B 0,C 180,E1 -16622.691,E2 -16622.691} C_VEL
LIN {X 0,Y 301.924,Z 218.453,A -85,B 0,C 180,E1 -16623.806,E2 -16623.806} C_VEL
LIN {X 0,Y 304.691,Z 235.25,A -85,B 0,C 180,E1 -16624.49,E2 -16624.49} C_VEL
LIN {X 0,Y 303.165,Z 293.945,A -85,B 0,C 180,E1 -16625.884,E2 -16625.884} C_VEL
LIN {X 0,Y 302.484,Z 304.644,A -85,B 0,C 180,E1 -16626.282,E2 -16626.282} C_VEL
LIN {X 0,Y 301.691,Z 313.742,A -85,B 0,C 180,E1 -16626.761,E2 -16626.761} C_VEL
LIN {X 0,Y 300.563,Z 324.101,A -85,B 0,C 180,E1 -16627.487,E2 -16627.487} C_VEL
LIN {X 0,Y 299.491,Z 333.235,A -85,B 0,C 180,E1 -16628.309,E2 -16628.309} C_VEL
LIN {X 0,Y 298.141,Z 342.227,A -85,B 0,C 180,E1 -16629.293,E2 -16629.293} C_VEL
LIN {X 0,Y 296.718,Z 350.952,A -85,B 0,C 180,E1 -16630.454,E2 -16630.454} C_VEL
LIN {X 0,Y 295.495,Z 358.346,A -85,B 0,C 180,E1 -16631.631,E2 -16631.631} C_VEL
LIN {X 0,Y 294.37,Z 365.291,A -85,B 0,C 180,E1 -16632.934,E2 -16632.934} C_VEL
LIN {X 0,Y 293.221,Z 371.767,A -85,B 0,C 180,E1 -16634.357,E2 -16634.357} C_VEL
LIN {X 0,Y 292.079,Z 378.304,A -85,B 0,C 180,E1 -16636.077,E2 -16636.077} C_VEL
LIN {X 0,Y 291.254,Z 382.805,A -85,B 0,C 180,E1 -16637.457,E2 -16637.457} C_VEL
LIN {X 0,Y 290.431,Z 388.299,A -85,B 0,C 180,E1 -16639.544,E2 -16639.544} C_VEL
LIN {X 0,Y 289.857,Z 392.625,A -85,B 0,C 180,E1 -16641.635,E2 -16641.635} C_VEL
LIN {X 0,Y 289.609,Z 394.994,A -85,B 0,C 180,E1 -16643.031,E2 -16643.031} C_VEL
LIN {X 0,Y 289.475,Z 396.912,A -85,B 0,C 180,E1 -16644.518,E2 -16644.518} C_VEL
LIN {X 0,Y 289.431,Z 399.245,A -85,B 0,C 180,E1 -16647.216,E2 -16647.216} C_VEL
LIN {X 0,Y 289.408,Z 399.835,A -85,B 0,C 180,E1 -16648.609,E2 -16648.609} C_VEL
LIN {X 0,Y 289.408,Z 399.835,A -85,B 0,C 180,E1 -16651.391,E2 -16651.391} C_VEL
LIN {X 0,Y 289.431,Z 399.245,A -85,B 0,C 180,E1 -16652.784,E2 -16652.784} C_VEL
LIN {X 0,Y 289.479,Z 396.795,A -85,B 0,C 180,E1 -16655.573,E2 -16655.573} C_VEL
LIN {X 0,Y 289.721,Z 393.843,A -85,B 0,C 180,E1 -16657.667,E2 -16657.667} C_VEL
LIN {X 0,Y 290.194,Z 389.853,A -85,B 0,C 180,E1 -16659.76,E2 -16659.76} C_VEL
LIN {X 0,Y 290.957,Z 384.722,A -85,B 0,C 180,E1 -16661.848,E2 -16661.848} C_VEL
LIN {X 0,Y 291.875,Z 379.46,A -85,B 0,C 180,E1 -16663.578,E2 -16663.578} C_VEL
LIN {X 0,Y 292.989,Z 373.144,A -85,B 0,C 180,E1 -16665.299,E2 -16665.299} C_VEL
LIN {X 0,Y 294.076,Z 367.194,A -85,B 0,C 180,E1 -16666.665,E2 -16666.665} C_VEL
LIN {X 0,Y 295.182,Z 360.265,A -85,B 0,C 180,E1 -16668.03,E2 -16668.03} C_VEL
LIN {X 0,Y 296.533,Z 352.087,A -85,B 0,C 180,E1 -16669.378,E2 -16669.378} C_VEL
LIN {X 0,Y 297.919,Z 343.578,A -85,B 0,C 180,E1 -16670.543,E2 -16670.543} C_VEL
LIN {X 0,Y 299.196,Z 334.865,A -85,B 0,C 180,E1 -16671.532,E2 -16671.532} C_VEL
LIN {X 0,Y 300.504,Z 325.11,A -85,B 0,C 180,E1 -16672.427,E2 -16672.427} C_VEL
LIN {X 0,Y 301.549,Z 315.029,A -85,B 0,C 180,E1 -16673.159,E2 -16673.159} C_VEL
LIN {X 0,Y 302.415,Z 305.518,A -85,B 0,C 180,E1 -16673.679,E2 -16673.679} C_VEL
LIN {X 0,Y 303.105,Z 295.208,A -85,B 0,C 180,E1 -16674.075,E2 -16674.075} C_VEL
LIN {X 0,Y 304.636,Z 234.178,A -85,B 0,C 180,E1 -16675.543,E2 -16675.543} C_VEL
LIN {X 0,Y 300.711,Z 212.324,A -85,B 0,C 180,E1 -16676.466,E2 -16676.466} C_VEL
LIN {X 0,Y 296.126,Z 191.965,A -85,B 0,C 180,E1 -16677.448,E2 -16677.448} C_VEL
LIN {X 0,Y 295.257,Z 189.155,A -85,B 0,C 180,E1 -16677.663,E2 -16677.663} C_VEL
LIN {X 0,Y 294.846,Z 186.954,A -85,B 0,C 180,E1 -16678.471,E2 -16678.471} C_VEL
LIN {X 0,Y 293.119,Z 177.876,A -85,B 0,C 180,E1 -16682.339,E2 -16682.339} C_VEL
LIN {X 0,Y 291.407,Z 169.73,A -85,B 0,C 180,E1 -16686.005,E2 -16686.005} C_VEL
LIN {X 0,Y 291.388,Z 169.661,A -85,B 0,C 180,E1 -16689.482,E2 -16689.482} C_VEL
LIN {X 0,Y 291.311,Z 169.7,A -85,B 0,C 180,E1 -16693.633,E2 -16693.633} C_VEL
LIN {X 0,Y 291.321,Z 169.7,A -85,B 0,C 180,E1 -16697.507,E2 -16697.507} C_VEL
LIN {X 0,Y 291.363,Z 169.683,A -85,B 0,C 180,E1 -16701.159,E2 -16701.159} C_VEL
LIN {X 0,Y 291.361,Z 169.677,A -85,B 0,C 180,E1 -16704.625,E2 -16704.625} C_VEL
LIN {X 0,Y 291.37,Z 169.687,A -85,B 0,C 180,E1 -16707.95,E2 -16707.95} C_VEL
LIN {X 0,Y 291.377,Z 169.677,A -85,B 0,C 180,E1 -16711.157,E2 -16711.157} C_VEL
LIN {X 0,Y 291.413,Z 169.664,A -85,B 0,C 180,E1 -16714.271,E2 -16714.271} C_VEL
LIN {X 0,Y 291.381,Z 169.687,A -85,B 0,C 180,E1 -16717.299,E2 -16717.299} C_VEL
LIN {X 0,Y 291.457,Z 169.649,A -85,B 0,C 180,E1 -16720.269,E2 -16720.269} C_VEL
LIN {X 0,Y 291.554,Z 169.661,A -85,B 0,C 180,E1 -16724.623,E2 -16724.623} C_VEL
LIN {X 0,Y 291.534,Z 169.642,A -85,B 0,C 180,E1 -16728.88,E2 -16728.88} C_VEL
LIN {X 0,Y 291.686,Z 169.622,A -85,B 0,C 180,E1 -16731.687,E2 -16731.687} C_VEL
LIN {X 0,Y 291.626,Z 169.657,A -85,B 0,C 180,E1 -16734.467,E2 -16734.467} C_VEL
LIN {X 0,Y 291.886,Z 169.599,A -85,B 0,C 180,E1 -16738.62,E2 -16738.62} C_VEL
LIN {X 0,Y 291.887,Z 169.595,A -85,B 0,C 180,E1 -16741.379,E2 -16741.379} C_VEL
LIN {X 0,Y 291.744,Z 169.635,A -85,B 0,C 180,E1 -16746.917,E2 -16746.917} C_VEL
LIN {X 0,Y 291.626,Z 169.621,A -85,B 0,C 180,E1 -16749.711,E2 -16749.711} C_VEL
LIN {X 0,Y 291.518,Z 169.671,A -85,B 0,C 180,E1 -16753.95,E2 -16753.95} C_VEL
LIN {X 0,Y 291.484,Z 169.666,A -85,B 0,C 180,E1 -16756.817,E2 -16756.817} C_VEL
LIN {X 0,Y 291.447,Z 169.649,A -85,B 0,C 180,E1 -16759.874,E2 -16759.874} C_VEL
LIN {X 0,Y 291.397,Z 169.684,A -85,B 0,C 180,E1 -16764.205,E2 -16764.205} C_VEL
LIN {X 0,Y 291.419,Z 169.657,A -85,B 0,C 180,E1 -16767.271,E2 -16767.271} C_VEL
LIN {X 0,Y 291.333,Z 169.695,A -85,B 0,C 180,E1 -16770.436,E2 -16770.436} C_VEL
LIN {X 0,Y 291.34,Z 169.674,A -85,B 0,C 180,E1 -16773.698,E2 -16773.698} C_VEL
LIN {X 0,Y 291.39,Z 169.689,A -85,B 0,C 180,E1 -16777.258,E2 -16777.258} C_VEL
LIN {X 0,Y 291.33,Z 169.678,A -85,B 0,C 180,E1 -16780.642,E2 -16780.642} C_VEL
LIN {X 0,Y 291.31,Z 169.694,A -85,B 0,C 180,E1 -16784.397,E2 -16784.397} C_VEL
LIN {X 0,Y 291.322,Z 169.642,A -85,B 0,C 180,E1 -16788.404,E2 -16788.404} C_VEL
LIN {X 0,Y 291.361,Z 169.687,A -85,B 0,C 180,E1 -16791.16,E2 -16791.16} C_VEL
LIN {X 0,Y 291.381,Z 169.657,A -85,B 0,C 180,E1 -16794.629,E2 -16794.629} C_VEL
LIN {X 0,Y 291.373,Z 169.691,A -85,B 0,C 180,E1 -16797.951,E2 -16797.951} C_VEL
LIN {X 0,Y 291.428,Z 169.827,A -85,B 0,C 180,E1 -16801.616,E2 -16801.616} C_VEL
LIN {X 0,Y 291.696,Z 170.932,A -85,B 0,C 180,E1 -16801.893,E2 -16801.893} C_VEL
LIN {X 0,Y 298.164,Z 182.952,A -85,B 0,C 180,E1 -16802.894,E2 -16802.894} C_VEL
LIN {X 0,Y 305.817,Z 193.62,A -85,B 0,C 180,E1 -16803.928,E2 -16803.928} C_VEL
LIN {X 0,Y 312.908,Z 201.762,A -85,B 0,C 180,E1 -16804.929,E2 -16804.929} C_VEL
LIN {X 0,Y 318.86,Z 208.209,A -85,B 0,C 180,E1 -16805.858,E2 -16805.858} C_VEL
LIN {X 0,Y 324.614,Z 214.288,A -85,B 0,C 180,E1 -16806.867,E2 -16806.867} C_VEL
LIN {X 0,Y 331.288,Z 220.922,A -85,B 0,C 180,E1 -16808.141,E2 -16808.141} C_VEL
LIN {X 0,Y 339.137,Z 228.332,A -85,B 0,C 180,E1 -16809.78,E2 -16809.78} C_VEL
LIN {X 0,Y 346.567,Z 234.931,A -85,B 0,C 180,E1 -16811.494,E2 -16811.494} C_VEL
LIN {X 0,Y 350.845,Z 238.399,A -85,B 0,C 180,E1 -16812.555,E2 -16812.555} C_VEL
LIN {X 0,Y 356.027,Z 242.823,A -85,B 0,C 180,E1 -16813.957,E2 -16813.957} C_VEL
LIN {X 0,Y 360.801,Z 246.482,A -85,B 0,C 180,E1 -16815.365,E2 -16815.365} C_VEL
LIN {X 0,Y 365.509,Z 250.364,A -85,B 0,C 180,E1 -16816.91,E2 -16816.91} C_VEL
LIN {X 0,Y 369.811,Z 253.164,A -85,B 0,C 180,E1 -16818.497,E2 -16818.497} C_VEL
LIN {X 0,Y 372.051,Z 254.669,A -85,B 0,C 180,E1 -16819.423,E2 -16819.423} C_VEL
LIN {X 0,Y 375.289,Z 257.587,A -85,B 0,C 180,E1 -16820.977,E2 -16820.977} C_VEL
LIN {X 0,Y 378.557,Z 259.876,A -85,B 0,C 180,E1 -16822.854,E2 -16822.854} C_VEL
LIN {X 0,Y 381.111,Z 261.225,A -85,B 0,C 180,E1 -16824.742,E2 -16824.742} C_VEL
LIN {X 0,Y 382.566,Z 261.76,A -85,B 0,C 180,E1 -16826.158,E2 -16826.158} C_VEL
LIN {X 0,Y 383.835,Z 262.318,A -85,B 0,C 180,E1 -16828.164,E2 -16828.164} C_VEL
LIN {X 0,Y 384.216,Z 262.461,A -85,B 0,C 180,E1 -16830,E2 -16830} C_VEL
LIN {X 0,Y 383.919,Z 262.382,A -85,B 0,C 180,E1 -16831.573,E2 -16831.573} C_VEL
LIN {X 0,Y 383.104,Z 261.923,A -85,B 0,C 180,E1 -16833.155,E2 -16833.155} C_VEL
LIN {X 0,Y 381.392,Z 261.375,A -85,B 0,C 180,E1 -16835.012,E2 -16835.012} C_VEL
LIN {X 0,Y 378.868,Z 260.056,A -85,B 0,C 180,E1 -16836.944,E2 -16836.944} C_VEL
LIN {X 0,Y 375.593,Z 257.806,A -85,B 0,C 180,E1 -16838.862,E2 -16838.862} C_VEL
LIN {X 0,Y 372.101,Z 254.738,A -85,B 0,C 180,E1 -16840.552,E2 -16840.552} C_VEL
LIN {X 0,Y 369.473,Z 252.943,A -85,B 0,C 180,E1 -16841.641,E2 -16841.641} C_VEL
LIN {X 0,Y 364.812,Z 249.849,A -85,B 0,C 180,E1 -16843.33,E2 -16843.33} C_VEL
LIN {X 0,Y 359.987,Z 245.743,A -85,B 0,C 180,E1 -16844.892,E2 -16844.892} C_VEL
LIN {X 0,Y 353.899,Z 241.155,A -85,B 0,C 180,E1 -16846.631,E2 -16846.631} C_VEL
LIN {X 0,Y 348.07,Z 236.103,A -85,B 0,C 180,E1 -16848.142,E2 -16848.142} C_VEL
LIN {X 0,Y 342.457,Z 231.34,A -85,B 0,C 180,E1 -16849.468,E2 -16849.468} C_VEL
LIN {X 0,Y 334.851,Z 224.421,A -85,B 0,C 180,E1 -16851.127,E2 -16851.127} C_VEL
LIN {X 0,Y 326.867,Z 216.55,A -85,B 0,C 180,E1 -16852.716,E2 -16852.716} C_VEL
LIN {X 0,Y 320.475,Z 210.048,A -85,B 0,C 180,E1 -16853.863,E2 -16853.863} C_VEL
LIN {X 0,Y 312.428,Z 201.297,A -85,B 0,C 180,E1 -16855.141,E2 -16855.141} C_VEL
LIN {X 0,Y 304.551,Z 191.987,A -85,B 0,C 180,E1 -16856.245,E2 -16856.245} C_VEL
LIN {X 0,Y 297.451,Z 181.749,A -85,B 0,C 180,E1 -16857.209,E2 -16857.209} C_VEL
LIN {X 0,Y 291.649,Z 170.78,A -85,B 0,C 180,E1 -16858.13,E2 -16858.13} C_VEL
LIN {X 0,Y 291.411,Z 169.75,A -85,B 0,C 180,E1 -16858.451,E2 -16858.451} C_VEL
LIN {X 0,Y 291.344,Z 169.687,A -85,B 0,C 180,E1 -16862.405,E2 -16862.405} C_VEL
LIN {X 0,Y 291.381,Z 169.657,A -85,B 0,C 180,E1 -16865.371,E2 -16865.371} C_VEL
LIN {X 0,Y 291.361,Z 169.687,A -85,B 0,C 180,E1 -16868.84,E2 -16868.84} C_VEL
LIN {X 0,Y 291.314,Z 169.643,A -85,B 0,C 180,E1 -16872.493,E2 -16872.493} C_VEL
LIN {X 0,Y 291.315,Z 169.697,A -85,B 0,C 180,E1 -16876.364,E2 -16876.364} C_VEL
LIN {X 0,Y 291.383,Z 169.678,A -85,B 0,C 180,E1 -16880.517,E2 -16880.517} C_VEL
LIN {X 0,Y 291.421,Z 169.684,A -85,B 0,C 180,E1 -16882.923,E2 -16882.923} C_VEL
LIN {X 0,Y 291.34,Z 169.674,A -85,B 0,C 180,E1 -16886.302,E2 -16886.302} C_VEL
LIN {X 0,Y 291.383,Z 169.683,A -85,B 0,C 180,E1 -16890.261,E2 -16890.261} C_VEL
LIN {X 0,Y 291.412,Z 169.668,A -85,B 0,C 180,E1 -16894.272,E2 -16894.272} C_VEL
LIN {X 0,Y 291.378,Z 169.688,A -85,B 0,C 180,E1 -16897.3,E2 -16897.3} C_VEL
LIN {X 0,Y 291.454,Z 169.647,A -85,B 0,C 180,E1 -16900.271,E2 -16900.271} C_VEL
LIN {X 0,Y 291.552,Z 169.667,A -85,B 0,C 180,E1 -16904.624,E2 -16904.624} C_VEL
LIN {X 0,Y 291.533,Z 169.641,A -85,B 0,C 180,E1 -16908.881,E2 -16908.881} C_VEL
LIN {X 0,Y 291.707,Z 169.622,A -85,B 0,C 180,E1 -16911.689,E2 -16911.689} C_VEL
LIN {X 0,Y 291.628,Z 169.658,A -85,B 0,C 180,E1 -16914.469,E2 -16914.469} C_VEL
LIN {X 0,Y 291.887,Z 169.595,A -85,B 0,C 180,E1 -16918.621,E2 -16918.621} C_VEL
LIN {X 0,Y 291.886,Z 169.599,A -85,B 0,C 180,E1 -16921.38,E2 -16921.38} C_VEL
LIN {X 0,Y 291.734,Z 169.633,A -85,B 0,C 180,E1 -16926.919,E2 -16926.919} C_VEL
LIN {X 0,Y 291.573,Z 169.626,A -85,B 0,C 180,E1 -16929.715,E2 -16929.715} C_VEL
LIN {X 0,Y 291.515,Z 169.668,A -85,B 0,C 180,E1 -16933.865,E2 -16933.865} C_VEL
